// TwinCAT 3 PLC project CEFPLC
// ProgramVersion: 3.1.4022.3
// libraries:
//   Tc2_Standard, * (Beckhoff Automation GmbH)
//   Tc2_System, * (Beckhoff Automation GmbH)
//   Tc2_Utilities, * (Beckhoff Automation GmbH)
//   Tc3_Database, * (Beckhoff Automation GmbH)
//   Tc3_EventLogger, * (Beckhoff Automation GmbH)
//   Tc3_Module, * (Beckhoff Automation GmbH)
//   VisuDialogs, * (System)
//   VisuSymbols,3.5.10.0,System
// project tree:
//   DUTs/ ST_ChamberAlarm.TcDUT, ST_ProgramListStruct.TcDUT, ST_ProgramStruct.TcDUT, ST_ScheduleStruct.TcDUT
//   FB/ fbCalculateSetpoint.TcPOU, scaleValue.TcPOU
//   / GlobalTextList.TcGTLO, PlcTask.TcTTO, ST_Record.TcDUT, Visualization Manager.TcVMO (not stored), VISU_TASK.TcTTO
//   GVLs/ GVL.TcGVL, IO_VARS.TcGVL
//   POUs/ AlarmLogger.TcPOU, DeleteOldData.TcPOU, Humidity.TcPOU, HumidityPID.TcPOU, HeaterDuty.TcPOU, TempPID.TcPOU, IO.TcPOU, OkToRun.TcPOU, MAIN.TcPOU, Watering.TcPOU
//   POUs/OLD NOT USED/ POU.TcPOU, fbGetNextLine.TcPOU, fbGetNextLineAfterMidnight.TcPOU, GetPreviousLine.TcPOU
//   POUs/Program Setpoints/ DatabaseStateMachine.TcPOU, DBConnector.TcPOU, QueryProgram.TcPOU
//   POUs/Scheduing/ fbGetCurrentProgramName.TcPOU, fbGetCurrentScheduleLine.TcPOU, fbGetFirstScheduleLine.TcPOU, fbGetNextScheduleLine.TcPOU, Scheduler.TcPOU
//   VISUs/ HMI_MAIN.TcVIS, OverviewScreen.TcVIS, GraphScreen.TcVIS, Settings.TcVIS, ProgramScreen.TcVIS, ImagePool.TcIPO (not stored), ManualMode.TcVIS, IO.TcVIS, Alarms.TcVIS, Watering.TcVIS
// real-time tasks:
//   TASK PlcTask: cycle T#10ms, priority 20, ADS port 350
//   TASK VISU_TASK: cycle T#50000us, priority 30, ADS port 351
// I/O:
//   DEVICE Device 2 (EtherCAT), AmsNetId 192.168.1.102.3.1
//     Term 1 (EK1100) [EK1100 EtherCAT Coupler (2A E-Bus)]
//       Term 2 (EL1008) [EL1008 8Ch. Dig. Input 24V, 3ms]
//       Term 3 (EL2008) [EL2008 8Ch. Dig. Output 24V, 0.5A]
//       Term 4 (EL2008) [EL2008 8Ch. Dig. Output 24V, 0.5A]
//       Term 5 (EL3064) [EL3064 4Ch. Ana. Input 0-10V]
//       Term 6 (EL4002) [EL4002 2Ch. Ana. Output 0-10V, 12bit]
//       Term 7 (EL9011) [EL9011 End Terminal]
// variable links:
//   CEFPLC/CEFPLC Instance <-> Device 2 (EtherCAT)/Term 1 (EK1100)/Term 3 (EL2008)
//     PlcTask Outputs/IO_VARS.HPS1 <-> Channel 4/Output
//     PlcTask Outputs/IO_VARS.HPS2 <-> Channel 5/Output
//     PlcTask Outputs/IO_VARS.HPS3 <-> Channel 6/Output
//     PlcTask Outputs/IO_VARS.MH1 <-> Channel 1/Output
//     PlcTask Outputs/IO_VARS.MH2 <-> Channel 2/Output
//     PlcTask Outputs/IO_VARS.MH3 <-> Channel 3/Output
//   CEFPLC/CEFPLC Instance <-> Device 2 (EtherCAT)/Term 1 (EK1100)/Term 4 (EL2008)
//     PlcTask Outputs/IO_VARS.ALARM <-> Channel 5/Output
//     PlcTask Outputs/IO_VARS.AUX1 <-> Channel 1/Output
//     PlcTask Outputs/IO_VARS.AUX2 <-> Channel 2/Output
//     PlcTask Outputs/IO_VARS.AUX3 <-> Channel 3/Output
//     PlcTask Outputs/IO_VARS.ENABLE <-> Channel 7/Output
//     PlcTask Outputs/IO_VARS.HEATERS <-> Channel 4/Output
//     PlcTask Outputs/IO_VARS.HUMVALVE <-> Channel 6/Output
//   CEFPLC/CEFPLC Instance <-> Device 2 (EtherCAT)/Term 1 (EK1100)/Term 5 (EL3064)
//     PlcTask Inputs/GVL.tempSensor <-> AI Standard Channel 1/Value
//     PlcTask Inputs/GVL.tempSensor2 <-> AI Standard Channel 3/Value
//     PlcTask Inputs/IO_VARS.HUM_SENS <-> AI Standard Channel 2/Value
//     PlcTask Inputs/IO_VARS.HUM_SENS2 <-> AI Standard Channel 4/Value
//   CEFPLC/CEFPLC Instance <-> Device 2 (EtherCAT)/Term 1 (EK1100)/Term 6 (EL4002)
//     PlcTask Outputs/IO_VARS.FANSPEED <-> AO Outputs Channel 2/Analog output
//     PlcTask Outputs/IO_VARS.GLYCOL_VALVE <-> AO Outputs Channel 1/Analog output

CONFIGURATION CEFPLC
    RESOURCE PLC ON TwinCAT3
        TASK PlcTask(INTERVAL := T#10ms, PRIORITY := 20);
        TASK VISU_TASK(INTERVAL := T#50000us, PRIORITY := 30);
        PROGRAM MAIN WITH PlcTask : MAIN;
        PROGRAM VisuElems_Visu_Prg WITH VISU_TASK : VisuElems.Visu_Prg;
    END_RESOURCE
END_CONFIGURATION

// ---- DUTs/ST_ChamberAlarm.TcDUT
TYPE ST_ChamberAlarm :
STRUCT
	dtTime:STRING(255);
	sAlarmText:STRING(255);
	
	
END_STRUCT
END_TYPE

// ---- DUTs/ST_ProgramListStruct.TcDUT
TYPE ST_ProgramListStruct :
STRUCT
	ID: LINT;
	Name: STRING(255);
END_STRUCT
END_TYPE

// ---- DUTs/ST_ProgramStruct.TcDUT
{attribute 'enable_dynamic_creation'}
TYPE ST_ProgramStruct :
STRUCT
	ID: LINT;
	name: STRING(255);
	ProgramID: LINT;
	iTime: LINT;
	Temperature: LREAL;
	humidity: LREAL;
	Light1: INT;
	Light2: INT;
	DO10: BOOL;
	DO11: BOOL;
END_STRUCT
END_TYPE

// ---- DUTs/ST_ScheduleStruct.TcDUT
TYPE ST_ScheduleStruct :
STRUCT
	ID: LINT;
	Sequence: LINT;
	ProgramID: LINT;
END_STRUCT
END_TYPE

// ---- ST_Record.TcDUT
TYPE ST_Record :
STRUCT

    nID        : LINT;
    dtTimestamp: DATE_AND_TIME;
    sName      : STRING;
    nSensor1   : LREAL;
    nSensor2   : LREAL;
END_STRUCT
END_TYPE

// ---- GVLs/GVL.TcGVL
{attribute 'qualified_only'}
VAR_GLOBAL
	

	TempControl: LREAL;
	iTempControl AT %Q*:INT;
	cycleTime: LREAL;
	
	tempSensor AT %I*: INT; 
	tempSensor2 AT %I*: INT; 
	
	Temp,Temp2: LREAL;
	Humidity,Humidity2:LREAL;

	
	reset: BOOL;

	fbLocalSystemTime:FB_LocalSystemTime;

	programURL: STRING(255);
	graphURL:STRING(255);
		
	manualMode:BOOL;
	bActiveAlarm:BOOL;
	bCriticalAlarm:BOOL;
	sAlarmText:STRING(255);
	sInfoText:STRING(255);
	
	
	
END_VAR

VAR_GLOBAL PERSISTENT
	KpCooling : LREAL := 10;
	KiCooling : LREAL := 550;
	KdCooling : LREAL := 0;
	KvCooling : LREAL := 800;
	
	KpHeating : LREAL := 3000;
	KiHeating : LREAL := 550;
	KdHeating: LREAL := 0;
	KvHeating : LREAL := 320;
	
	KpHumidity : LREAL := 1;
	KiHumidity : LREAL := 1;
	KdHumidity: LREAL := 0;
	KvHumidity : LREAL := 1;
	
	CurrentProgram: LINT;
	CurrentProgramName:STRING(255);
	NextProgram: LINT;
	FirstProgram:LINT;
	ScheduleSequence:LINT;

	TempAlarmHigh:LREAL:=50;
	TempAlarmLow:LREAL:=4;
	
	TempCalibrationLimit:REAL:=10;//in percent
	HumCalibrationLimit:REAL:=10;//in percent
	//Don't change this without also changing
	//iMax in AlarmLogger
	aAlarms:ARRAY[0..15] OF ST_ChamberAlarm;
	
	okToRun:BOOL;
	iState:INT;
	
	
	
	//Setpoint variable declariations
	Light1Max:INT:=2; //Max light level
	Light1Level:INT; //Current light level
	Light1Percent:REAL; //Current light level in percent of max
	Light1Stepmode:BOOL;
	
	Light2Max:INT:=2; //Max light level
	Light2Level:INT; //Current light level
	Light2Percent:REAL; //Current light level in percent of max
	Light2Stepmode:BOOL;
	
	TempSetpoint: LREAL;
	TempStepmode: BOOL;
	
	HumiditySetpoint:LREAL;
	HumidityStepmode:BOOL;
	
	
	///HMI VARS
	HMIPowerButton:BOOL;
	HMIFanSpeed:INT;
	HMIWateringStartHour:DWORD;
	HMIWateringStartMinute:DWORD;
	HMIWateringTimeSeconds:DWORD;
	
	//Watering
	wateringDays: ARRAY[0..6] OF BOOL; //if element 0 is True, then water on Sunday, if element 1 is true, water on Monday. etc
	watertingTime:TIME;//How long to water
	watertingStart:TOD;//When to start watering
END_VAR

// ---- GVLs/IO_VARS.TcGVL
{attribute 'qualified_only'}
VAR_GLOBAL
	
PRESSURE_SENSE AT %I*:BOOL;
HUM_SENS,HUM_SENS2 AT %I*:INT;


ENABLE AT %Q*:BOOL;
MH1,MH2,MH3 AT %Q*:BOOL;
HPS1,HPS2,HPS3 AT %Q*:BOOL;
AUX1,AUX2,AUX3,ALARM AT %Q*:BOOL; 
HEATERS AT %Q*:BOOL;

HUMVALVE AT %Q*:BOOL;

GLYCOL_VALVE AT %Q*:INT;

END_VAR

VAR_GLOBAL PERSISTENT
	FANSPEED AT %Q*:INT;
END_VAR

// ---- POUs/MAIN.TcPOU
PROGRAM MAIN


VAR

	GETCPUCOUNTER: GETCPUCOUNTER; //CPU tick function block definition
	previous_low_ticks,low_ticks,high_ticks: UDINT; //Vars to hold the cpu tick count
	
	
	test: DINT; //I don't know what this is
	sqlResult : WSTRING(255);//I don't think we need this anymore either
	bsqlError: BOOL;//same ehere
	
	numberOfLinesOut: LINT; //and here
	Scaled_control: LREAL;//this moved too

	fbTON: TON := (PT := TIME#1S0MS); //PID TON TIMER.
	restartTime: TON := (PT := TIME#60S0MS);//AUTO RESTART TIMER

	

	getHost: FB_GetHostName; //Get host name function block definition
	myName: STRING(255); //Var to hold host name. If the host name is more than 255 chars you're doing something wrong.
	
	FB_WritePersistentData: FB_WritePersistentData;
	GETSYSTEMTIME:GETSYSTEMTIME;
END_VAR

/////////////////////////////////////////////////////////////
//CALCULATE CYCLE TIME FOR PLC
previous_low_ticks := low_ticks;
//GETCPUCOUNTER(cpuCntLoDW=> low_ticks, cpuCntHiDW=> high_ticks);
GETSYSTEMTIME(timeLoDW=> low_ticks, timeHiDW=> high_ticks);
//low ticks is a 64 bit int and rolls over into high ticks once in a while. So we make sure we're not calculating the overflow
IF previous_low_ticks < low_ticks THEN 
	GVL.cycleTime := UDINT_TO_LREAL(low_ticks-previous_low_ticks)*0.000000100;//Each tick is 100ns
END_IF

/////////////////////////////////////////////////////////////
//GET HOST NAME AND CONCAT URLS FOR HMI SCREENS
//we need the hostname because "localhost" doesn't work if
//you're connected remotely, duh
getHost(bExecute:= TRUE, sHostName=>myName );
GVL.programURL:=CONCAT('http://',myName);
GVL.programURL:=CONCAT(GVL.programURL,':8050');
GVL.graphURL:=CONCAT('http://',myName);
GVL.graphURL:=CONCAT(GVL.graphURL,':8050/graph');
/////////////////////////////////////////////////////////////
//VARIOUS PROGRAMS THAT NEED TO RUN EVERY CYCLE
IO(); //Input/Output tasks and calculations
Humidity();
HeaterDuty();
OkToRun();//Alarms
fbTON();//Timer for some functions that we don't want to run every cycle
restartTime();//Timer for auto restart in the event of an error. Set to 60 seconds
AlarmLogger();//Log alarms (if any)
GVL.fbLocalSystemTime(sNetID:= '', bEnable:= TRUE, dwCycle:= 1);//Get the current date and time

/////////////////////////////////////////////////////////////
//VARIOUS PROGRAMS THAT DO NOT RUN EVERY CYCLE

IF fbTON.Q=TRUE THEN //when the timer is true (every 1 second)
	TempPID();//Run the PIDs
	HumidityPID();
	fbTON.IN:=FALSE; //reset the timer
	FB_WritePersistentData(NETID:='', PORT:=851, START:=TRUE, TMOUT:=T#1S ); //Write persistent data 
	Scheduler();//Checking/setting program schedule
	DeleteOldData();
	Watering();
ELSE
	fbTON.IN:=TRUE; //If the timer is not true...keep timing until it is!
END_IF
/////////////////////////////////////////////////////////////
//MAIN STATE MACHINE
CASE GVL.iState OF
	//STARTUP
	0:
		
		GVL.reset:=TRUE; //RESET THE PID MEMORY BEFORE STARTING. THIS IS IMPORTANT.
		Scheduler.resetSchedule:=TRUE; //RESET THE SCHEDULE BACK TO THE BEGINNING 
		
		IF GVL.sInfoText='' THEN//If the info text is blank, give the user a hint to get started
			GVL.sInfoText:='Setup programs & settings then Start';
		END_IF
		//Check if user presses start button	
		IF GVL.HMIPowerButton=TRUE THEN

			DatabaseStateMachine.bStepStart:=TRUE; //STEP START MEANS THE FIRST SETPOINT WILL BE STEPPED TO GET STARTED. MORE INFO IN DOCS
			DatabaseStateMachine(); //ALL SETPOINTS ARE CONTROLLED BY THE DATABASE STATE MACHINE. THIS PROGRAM IS IMPORTANT.
			
			GVL.sAlarmText:='Wait for Startup...';
			GVL.sInfoText:='Checking Setpoints...';
			IF DatabaseStateMachine.allOutputsSet=TRUE AND GVL.okToRun=TRUE THEN //Once everything is set, we can move on to the next state
				GVL.iState:=1;
				
			END_IF
	
		END_IF
		
		IF GVL.manualMode THEN
			GVL.iState:=254;
		END_IF
	
	1:
		//Runninng

		GVL.reset:=FALSE; //Don't reset the PID while running
		
		DatabaseStateMachine.bStepStart:=FALSE;//Don't need step start because we're already running!
		DatabaseStateMachine();//Running the statemachine....
		GVL.sInfoText:=''; //Everything is good! We don't need any info text
		
		//Check if shutdown
		//Lots of things can make OktoRun False. Check the sub program and the Docs.
		IF GVL.okToRun=FALSE THEN 
			GVL.iState:=2;
		END_IF
		
	2:
	//Shutdown
	
	IF GVL.bCriticalAlarm=FALSE THEN //If shutdown with no error
		
		GVL.iState:=0;

		
	ELSIF GVL.bCriticalAlarm=TRUE THEN//If shutdown WITH error

		restartTime.IN:=TRUE;
		GVL.sInfoText:='Acknowledge alarm or wait for auto restart';
		IF restartTime.Q THEN //Try restarting after the timer has elapsed
			GVL.HMIPowerButton:=TRUE;
			GVL.bCriticalAlarm:=FALSE;
			restartTime.IN:=FALSE;
			GVL.iState:=1;
			GVL.sInfoText:='Error occured...restarting';
		ELSIF GVL.bActiveAlarm=FALSE THEN //Clear error if the user has pressed the acknowledge alarm button
			restartTime.IN:=FALSE;
			GVL.bCriticalAlarm:=FALSE;
			GVL.iState:=0;
			GVL.sInfoText:='Alarm acknowledged, please manually restart program ';
		END_IF

	END_IF
	254:
	//Manual Mode
	//Just don't do anything until the user exits manual mode
		GVL.sAlarmText:='MANUAL MODE ACTIVE';
		IF GVL.manualMode=FALSE THEN
			GVL.iState:=2;
		END_IF
	
END_CASE

END_PROGRAM

// ---- POUs/IO.TcPOU
PROGRAM IO
VAR


	Scaled_control: LREAL;

END_VAR


	

GVL.Temp := 0.010071*INT_TO_LREAL(GVL.tempSensor) - 39.996;//See documentation for sensor
GVL.Humidity := (INT_TO_LREAL(IO_VARS.HUM_SENS)/3.2767)*100/5000;

GVL.Temp2 := 0.010071*INT_TO_LREAL(GVL.tempSensor2) - 39.996;//See documentation for sensor
GVL.Humidity2 := (INT_TO_LREAL(IO_VARS.HUM_SENS2)/3.2767)*100/5000;

IO_VARS.ALARM:=GVL.bCriticalAlarm;//alarm buzzer


//Check this variable just to make sure we don't break anything
IF GVL.HMIFanSpeed>100 THEN
	GVL.HMIFanSpeed:=100;
END_IF

IF GVL.HMIFanSpeed<0 THEN
	GVL.HMIFanSpeed:=0;
END_IF

IO_VARS.FANSPEED := REAL_TO_INT(16384*-50*LOG(0.00001*(63949-630*GVL.HMIFanSpeed))/100);//Scaling. outout is nonlinear for this board. Equation is x = -50 log(.00001(63949 - 630 y))
	
IF IO_VARS.FANSPEED>16385 THEN
	IO_VARS.FANSPEED:=16385;//DO NOT EXCEED 5 VOLTS FOR THAT CONTROL BOARD
END_IF

IF IO_VARS.FANSPEED<3276 THEN
	IO_VARS.FANSPEED:=3276;//IT'S DANGERIOUS TO RUN THE CHAMBER WITH THE FANS COMPLETELY OFF
END_IF


IF GVL.manualMode=FALSE THEN
	
	//Set the valve state
	IO_VARS.GLYCOL_VALVE:=GVL.iTempControl;
	
	IO_VARS.AUX1:=Watering.waterOn;//Watering bound to aux 1
	
	//If the output of the pulse timer is true, turn on the heater valve
	IO_VARS.HEATERS:=HeaterDuty.HeatersON;
	
	//If the output of the pulse timer is true, turn on the humidity valve
	IO_VARS.HUMVALVE:=Humidity.HumidityON;
		
	////////////MAPPING METAL HALIDE LIGHTS/////////////
	IF GVL.Light1Level=0 THEN
		IO_VARS.MH1:=0;
		IO_VARS.MH2:=0;
		IO_VARS.MH3:=0;
	ELSIF  GVL.Light1Level=1 THEN
		IO_VARS.MH1:=1;
		IO_VARS.MH2:=0;
		IO_VARS.MH3:=0;
	ELSIF  GVL.Light1Level=2 THEN
		IO_VARS.MH1:=1;
		IO_VARS.MH2:=1;
		IO_VARS.MH3:=0;
	ELSIF  GVL.Light1Level=3 THEN
		IO_VARS.MH1:=1;
		IO_VARS.MH2:=1;
		IO_VARS.MH3:=1;
	END_IF
	
	////////////MAPPING HIGH PRESSURE SODIUM LIGHTS/////////////
	IF GVL.Light2Level=0 THEN
		IO_VARS.HPS1:=0;
		IO_VARS.HPS2:=0;
		IO_VARS.HPS3:=0;
	ELSIF  GVL.Light2Level=1 THEN
		IO_VARS.HPS1:=1;
		IO_VARS.HPS2:=0;
		IO_VARS.HPS3:=0;
	ELSIF  GVL.Light2Level=2 THEN
		IO_VARS.HPS1:=1;
		IO_VARS.HPS2:=1;
		IO_VARS.HPS3:=0;
	ELSIF  GVL.Light2Level=3 THEN
		IO_VARS.HPS1:=1;
		IO_VARS.HPS2:=1;
		IO_VARS.HPS3:=1;
	END_IF
	
END_IF

END_PROGRAM

// ---- POUs/Humidity.TcPOU
PROGRAM Humidity
VAR
	
	fbTON: TON; // TON TIMER.
	
	fbTP: TP;

	pulseDuration: TIME:=TIME#2S;
END_VAR

VAR_OUTPUT
	
HumidityON:BOOL;
	


END_VAR

//This program pulses the humidity for a certain number of seconds based on the PID output

//This timer determines how often to pulse, and the max length of the pulse
//In other words, we're making a Duty Cycle
fbTON(PT := TIME#30S0MS);

//Run the pulse timer
fbTP();

//If the output of the pulse timer is true, turn on the humidity valve
HumidityON:=fbTP.Q;


//Don't worry about negative values
IF HumidityPID.output >=0 THEN
	
	//Convert the output to a time (in milliseconds)
	pulseDuration:=LREAL_TO_TIME(HumidityPID.output);
	
	//Don't pulse anything shorter than 500ms.
	//It's bad for the relay & valve
	IF pulseDuration<TIME#500MS THEN
		pulseDuration:=TIME#0MS;
	END_IF
	
	//If the durataion is greater than the max duration
	//Just turn it on and leave it on
	IF pulseDuration>fbTON.PT THEN
		HumidityON:=TRUE;
	ELSE
	
		IF fbTON.Q=TRUE THEN //when the timer is true 
			fbTP(IN:=TRUE, PT:=pulseDuration);//set the pulse length
			fbTON.IN:=FALSE;//Reset the timer funtion
		ELSE
			fbTON.IN:=TRUE; //If the timer is not true...keep timing until it is!
			fbTP.IN:=FALSE;//reset the pulse function
		END_IF
			
	END_IF

END_IF

END_PROGRAM

// ---- POUs/HumidityPID.TcPOU
PROGRAM HumidityPID
VAR
	
	PID: FB_BasicPID;
	bReset: BOOL;
	
	AH: LREAL;
	AHSetpoint: LREAL;
	
	//Constants for air as an ideal gas to calculate absolute humidity in g/m^3
	Tn:LREAL:=240.7263;
	m:LREAL:=7.591386;
	A:LREAL:=6.116441;
END_VAR

VAR_OUTPUT
	output: LREAL;
END_VAR

//Convert realative humidity to absolute humidity in grams per cubic meter
AH:= A*EXPT	(10,m*GVL.Temp/(GVL.Temp+Tn))*(GVL.Humidity/100)*100*2.16679/(273.15+GVL.Temp);
AHSetpoint:= A*EXPT(10,m*GVL.TempSetpoint/(GVL.TempSetpoint+Tn))*(GVL.HumiditySetpoint/100)*100*2.16679/(273.15+GVL.TempSetpoint);

//Run pid loop
PID(
	fSetpointValue:=AHSetpoint,
	fActualValue:=AH, 
	bReset:=bReset, 
	fCtrlCycleTime:=1, 
	fKp:=GVL.KpHumidity, 
	fTn:=GVL.KiHumidity, 
	fTv:=GVL.KvHumidity, 
	fTd:=GVL.KdHumidity, 
	fCtrlOutput=>output);
	
	
//Since there's no dehumidification on this chamber
//Just reset the PID back to 0 if the output is negative
IF output<0 THEN
	output:=0;
	bReset:=TRUE;
ELSIF GVL.reset =  TRUE THEN
	bReset:=TRUE;
ELSE
	bReset:=FALSE;
END_IF

END_PROGRAM

// ---- POUs/Watering.TcPOU
PROGRAM Watering
VAR
	
	trigger:F_TRIG;
	waterTimer:TON;
	waterOn:BOOL;
	dtTime:DT;
	todTime:TOD;

END_VAR


GVL.watertingTime:=DWORD_TO_TIME(GVL.HMIWateringTimeSeconds*1000);//in ms
GVL.watertingStart:=DWORD_TO_TOD((GVL.HMIWateringStartHour*60 + GVL.HMIWateringStartMinute)*60*1000);//also in ms



dtTime:=SYSTEMTIME_TO_DT(GVL.fbLocalSystemTime.systemTime);
todTime:=DT_TO_TOD(dtTime);
waterTimer(PT:=GVL.watertingTime);

IF GVL.wateringDays[GVL.fbLocalSystemTime.systemTime.wDayOfWeek]=TRUE THEN
	IF todTime>=GVL.watertingStart AND todTime<=(GVL.watertingStart+GVL.watertingTime) THEN
		waterOn:=TRUE;
	ELSE
		waterOn:=FALSE;
	END_IF
END_IF

END_PROGRAM

// ---- POUs/HeaterDuty.TcPOU
PROGRAM HeaterDuty
VAR
	
	fbTON: TON; // TON TIMER.
	
	fbTP: TP;

	pulseDuration: TIME:=TIME#2S;
END_VAR

VAR_OUTPUT
	
HeatersON:BOOL;
	
END_VAR

//This program pulses the heaters for a certain number of seconds based on the PID output

//This timer determines how often to pulse, and the max length of the pulse
//In other words, we're making a Duty Cycle
fbTON(PT := TIME#30S0MS);

//Run the pulse timer
fbTP();

//If the output of the pulse timer is true, turn on the heater valve
HeatersON:=fbTP.Q;


//Don't worry about negative values
IF TempPID.HeatingOutput >=0 THEN
	
	//Convert the output to a time (in milliseconds)
	pulseDuration:=LREAL_TO_TIME(TempPID.HeatingOutput);
	
	//Don't pulse anything shorter than 500ms.
	//It's bad for the relay
	IF pulseDuration<TIME#500MS THEN
		pulseDuration:=TIME#0MS;
	END_IF
	
	//If the durataion is greater than the max duration
	//Just turn it on and leave it on
	IF pulseDuration>fbTON.PT THEN
		HeatersON:=TRUE;
	ELSE
	
		IF fbTON.Q=TRUE THEN //when the timer is true 
			fbTP(IN:=TRUE, PT:=pulseDuration);//set the pulse length
			fbTON.IN:=FALSE;//Reset the timer funtion
		ELSE
			fbTON.IN:=TRUE; //If the timer is not true...keep timing until it is!
			fbTP.IN:=FALSE;//reset the pulse function
		END_IF
			
	END_IF

END_IF

END_PROGRAM

// ---- POUs/TempPID.TcPOU
PROGRAM TempPID
VAR
	
	PIDCooling: FB_BasicPID;
	PIDHeating: FB_BasicPID;
	bResetCooling: BOOL;
	bResetHeat: BOOL;
END_VAR

VAR_OUTPUT
	CoolingOutput: LREAL;
	HeatingOutput: LREAL;
END_VAR



//Run pid loop
PIDCooling(
	fSetpointValue:=GVL.TempSetpoint,
	fActualValue:=GVL.Temp, 
	bReset:=bResetCooling, 
	fCtrlCycleTime:=1, 
	fKp:=GVL.KpCooling, 
	fTn:=GVL.KiCooling, 
	fTv:=GVL.KvCooling, 
	fTd:=GVL.KdCooling);



PIDHeating(
	fSetpointValue:=GVL.TempSetpoint,
	fActualValue:=GVL.Temp, 
	bReset:=bResetHeat, 
	fCtrlCycleTime:=1, 
	fKp:=GVL.KpHeating, 
	fTn:=GVL.KiHeating, 
	fTv:=GVL.KvHeating, 
	fTd:=GVL.KdHeating);
	
//Reset the PID back to 0 if the output is out of range
IF  PIDCooling.fCtrlOutput>50 THEN
	bResetCooling:=TRUE;
ELSIF GVL.reset =  TRUE THEN
	bResetCooling:=TRUE;
ELSE
	bResetCooling:=FALSE;
	CoolingOutput:=PIDCooling.fCtrlOutput*-105+14089; //<----important scaling function because the old staefa valves are weird. See documentation for siemens ZM-101A
END_IF

//Reset the PID back to 0 if the output is out of range
IF PIDHeating.fCtrlOutput<-30000 THEN
	bResetHeat:=TRUE;
ELSIF GVL.reset =  TRUE THEN
	bResetHeat:=TRUE;
ELSE
	bResetHeat:=FALSE;
	HeatingOutput:=PIDHeating.fCtrlOutput;//No need to scale the heater output. Just use PID constants
END_IF

//If there is more than 5% cooling demand, turn off the heaters completely. (i.e. don't waste energy)
IF PIDCooling.fCtrlOutput<-5 THEN
	HeatingOutput:=0;
END_IF

//Scale temp signal for analog out to avoid overflows/negative numbers
IF CoolingOutput>=32767 THEN
	GVL.iTempControl :=32767;
ELSIF CoolingOutput <=0 THEN
	GVL.iTempControl :=0;
ELSE
	GVL.iTempControl := LREAL_TO_INT(CoolingOutput);
END_IF

IF HeatingOutput>=30000 THEN
	HeatingOutput :=30000;
ELSIF HeatingOutput <=0 THEN
	HeatingOutput :=0;
ELSE
	HeatingOutput := HeatingOutput;
END_IF

END_PROGRAM

// ---- POUs/OkToRun.TcPOU
PROGRAM OkToRun
VAR

	alarmTimeout: TON := (PT := TIME#11S0MS);
	
END_VAR

alarmTimeout();

//HARD CODED UPPER AND LOWER LIMITS
IF GVL.Temp > 50 THEN
		GVL.bCriticalAlarm:=TRUE;
		IO_VARS.ENABLE:=FALSE;
		GVL.sAlarmText:='Critical High Temp Alarm';
	END_IF
IF GVL.Temp < 0 THEN
	GVL.bCriticalAlarm:=TRUE;
	IO_VARS.ENABLE:=FALSE;
	GVL.sAlarmText:='Critical Low Temp Alarm';
END_IF



//If not in manual mode
IF GVL.manualMode=FALSE THEN
	
	//If running
	IF GVL.iState=1 THEN

	
		//Temperature Alarm Logic for STEP MODE
		IF GVL.TempStepmode THEN
			IF GVL.iState=1 AND GVL.Temp > (GVL.TempAlarmHigh) THEN
				GVL.bCriticalAlarm:=TRUE;
				GVL.sAlarmText:='High Temp Alarm';
			END_IF
			IF GVL.iState=1 AND GVL.Temp < (GVL.TempAlarmLow) THEN
				GVL.bCriticalAlarm:=TRUE;
				GVL.sAlarmText:='Low Temp Alarm';
			END_IF
		END_IF
		
		//Temperature alarm logic for RAMP MODE
		IF GVL.TempStepmode=FALSE THEN
			IF GVL.iState=1 AND GVL.Temp > (GVL.TempSetpoint+GVL.TempAlarmHigh) THEN
				GVL.bCriticalAlarm:=TRUE;
				GVL.sAlarmText:='High Temp Alarm';
			END_IF
			IF GVL.iState=1 AND GVL.Temp < (GVL.TempSetpoint-GVL.TempAlarmLow) THEN
				GVL.bCriticalAlarm:=TRUE;
				GVL.sAlarmText:='Low Temp Alarm';
			END_IF
		END_IF
		
		//Schedule Alarms
		//If the user deletes the current program or changes the schedule in an incorrect way, 
		//Tell them they messed up
		//This could also happen if there are database errors
		IF fbGetCurrentScheduleLine.sSeverity="No Error" AND fbGetCurrentScheduleLine.iLines=0 THEN
			alarmTimeout.IN:=TRUE;
			IF alarmTimeout.Q=TRUE THEN
				GVL.sAlarmText:='Error getting current program. Check schedule and programs';
				GVL.bCriticalAlarm:=TRUE;
				alarmTimeout.IN:=FALSE;
				
			END_IF
				
		ELSE

			alarmTimeout.IN:=FALSE;
			
		END_IF
		//Temperature sensor alarm
		IF ABS((GVL.Temp-GVL.Temp2)*100/GVL.Temp)>GVL.TempCalibrationLimit THEN
				GVL.sAlarmText:='Temperature Sensor Error.';
				GVL.bCriticalAlarm:=TRUE;
		END_IF
		
		//Humidity sensor alarm
		IF ABS((GVL.Humidity-GVL.Humidity2)*100/GVL.Humidity)>GVL.HumCalibrationLimit THEN
				GVL.sAlarmText:='Humidity Sensor Error.';
				GVL.bCriticalAlarm:=TRUE;
		END_IF
		

	END_IF
	
	

END_IF	

//OK TO RUN IF THERE ARE NO ERRORS
IF GVL.bCriticalAlarm=FALSE AND GVL.HMIPowerButton=TRUE THEN
	GVL.okToRun:=TRUE;
	GVL.sAlarmText:='Running No Alarm';
	IO_VARS.ENABLE:=TRUE;
ELSIF GVL.bCriticalAlarm=FALSE AND GVL.HMIPowerButton=FALSE AND IO_VARS.ENABLE=FALSE THEN
	GVL.sAlarmText:='Not Running No Alarm';
ELSE
	GVL.okToRun:=FALSE;
	IF GVL.manualMode=FALSE THEN
		IO_VARS.ENABLE:=FALSE;
	END_IF
	
	GVL.HMIPowerButton:=FALSE;
END_IF

END_PROGRAM

// ---- POUs/Scheduing/fbGetCurrentScheduleLine.TcPOU
PROGRAM fbGetCurrentScheduleLine

VAR_OUTPUT
	arrRecords: ST_ScheduleStruct;
	sSeverity: WSTRING(255);
	bError :BOOL;

	iLines: UDINT;
END_VAR
VAR
	STProgram: ST_ProgramStruct;
	now : TIMESTRUCT;
	nowMinutes : LINT;
	
	previousMinute: LINT;
	
	fbTON: TON := (PT := TIME#10S0MS);

	

	
	fbPLCDBRead : FB_PLCDBRead(sNetID:='',tTimeout:=T#5S);
	fbSqlCommand : FB_SQLCommand(sNetID := '', tTimeout := T#5S);
	
	
	intTime: DINT;
	todTime: TOD;

	sCmd: STRING(255):='SELECT * FROM [Schedule] ORDER BY [Sequence] ASC';

	dIntSqlResult: DINT;
	fbSQLDatabase: FB_SQLDatabase(sNetID:='', tTimeout:=T#10S);
	fbSQLResult: FB_SQLResult(sNetID:='', tTimeout:=T#10S);
	result: I_TcResultEvent;


	iState: INT;
END_VAR

//Build command



sCmd :=CONCAT('SELECT * FROM [Schedule] WHERE [Sequence]=',LINT_TO_STRING(GVL.ScheduleSequence));

//State machine
CASE iState OF
0:
//IDLE
fbTON(PT := TIME#3S0MS);
IF fbTON.Q=TRUE THEN
	iState:=1;
	fbTON.IN:=FALSE;
	bError := FALSE; 
ELSE
	fbTON.IN:=TRUE;
END_IF
//Connect
1:
	IF fbSqlDatabase.Connect(1) THEN
		IF fbSqlDatabase.bError THEN
			iState := 255;
			result := fbSqlDatabase.ipTcResultEvent;
			sSeverity := result.Text;
			bError := TRUE; 		
		ELSE
			//If sucessful, point the connection to the sql command function
			fbSqlDatabase.CreateCmd(ADR(fbSqlCommand));
			iState := 2;
		END_IF
	END_IF
2:
//Send the sql command
	IF fbSQLCommand.ExecuteDataReturn(ADR(sCmd), SIZEOF(sCmd), ADR(fbSqlResult)) THEN
		IF fbSQLCommand.bError THEN
			iState := 255;
			result := fbSQLCommand.ipTcResultEvent;
			sSeverity := result.Text;
			bError := TRUE;
		ELSE
			iState := 3; 
			iLines:=fbSqlResult.nDataCount;
		END_IF
	END_IF
		
3:
//Read the sql result
	IF fbSqlResult.Read(0, 1, ADR(arrRecords), SIZEOF(arrRecords), TRUE, TRUE) THEN
		IF fbSqlResult.bError THEN
			result := fbSqlResult.ipTcResultEvent;
			sSeverity := result.Text;
			iState:=255;
			bError := TRUE;
		ELSE 
			iState:=4;
			
			result := fbSqlResult.ipTcResultEvent;
			sSeverity := result.Text;
		END_IF
	

	END_IF
4:
	IF 	fbSqlDatabase.Disconnect() THEN
		bError := FALSE;
		iState:=0;
	END_IF
255:
	IF 	fbSqlDatabase.Disconnect() THEN
		iState:=0;	
		bError := TRUE;
		result := fbSqlResult.ipTcResultEvent;
		sSeverity := result.Text;

	END_IF
	
END_CASE

END_PROGRAM

// ---- POUs/AlarmLogger.TcPOU
PROGRAM AlarmLogger
VAR
	iCounter:DINT;
	iMax:DINT;
	alarmTrigger: R_TRIG; 
END_VAR

alarmTrigger(CLK := GVL.bCriticalAlarm);

IF alarmTrigger.Q THEN
	//Shift the whole array by 1 so we can enter the new alarm in the first element
	iCounter:=0;
	
	//Max number of alarms
	//Depends on the array size of GVL.aAlarms
	iMax:=15;
	
	FOR iCounter:=iMax TO 0 BY -1 DO //Notice we're counting backwards so the last element goes away, and the first element is now empty
		
		IF iCounter<>iMax THEN
			GVL.aAlarms[iCounter+1]:=GVL.aAlarms[iCounter];
		END_IF	

	END_FOR

	GVL.aAlarms[0].sAlarmText:=GVL.sAlarmText;
	GVL.aAlarms[0].dtTime:=SYSTEMTIME_TO_STRING(GVL.fbLocalSystemTime.systemTime);
	
	GVL.bActiveAlarm:=TRUE; //An alarm is now active and will remain that way until the user acknowledges it

END_IF

END_PROGRAM

// ---- POUs/Scheduing/Scheduler.TcPOU
PROGRAM Scheduler
VAR_INPUT
	resetSchedule:BOOL:=TRUE;
END_VAR
VAR
	
	
	
	ScheduleLine:ST_ScheduleStruct;
	sqlResult:WSTRING(255);
	bError:BOOL;
	iLines:UDINT;
	iState:INT;

	lastDate: TIMESTRUCT;
END_VAR


//Run all these programs to get the next line, first line, and current line in the schedule using database queries
fbGetNextScheduleLine();
fbGetCurrentScheduleLine();
fbGetFirstScheduleLine();
fbGetCurrentProgramName();
GVL.CurrentProgramName:=fbGetCurrentProgramName.arrRecords.Name;

CASE iState OF

0:
iState:=1;
//IDLE...nothing here yet

	
1:
	//If we want to reset the schedule to the beginning
	IF resetSchedule=TRUE THEN
		
		
		IF fbGetFirstScheduleLine.sSeverity="No Error" THEN //If there is no error when we try and get the first line in the schedule
			GVL.CurrentProgram:=fbGetFirstScheduleLine.arrRecords.ProgramID;
			//We need to initialize the next program to something. So we just set it to the current program
			GVL.NextProgram:=fbGetFirstScheduleLine.arrRecords.ProgramID;
			//The sequence is an integer that determines the order to run the programs. 1->2-->3 etc
			//This is set by the user in the interface. Here we just read the value
			GVL.ScheduleSequence:=fbGetFirstScheduleLine.arrRecords.Sequence;
			
			//OK we reset the schedule, set that to false now
			resetSchedule:=FALSE;
			
			//Timestamp when it happened so we know when a full day has passed
			lastDate := GVL.fbLocalSystemTime.systemTime;
		END_IF
	ELSIF resetSchedule=FALSE THEN
		//Check for the current and next programs in the schedule
		
		//While running, check to see if the schedule has changed
		//If the schedule has changed, then change the program to match
		IF fbGetCurrentScheduleLine.arrRecords.ProgramID<>GVL.CurrentProgram AND fbGetCurrentScheduleLine.sSeverity="No Error" AND fbGetCurrentScheduleLine.iLines<>0	THEN
			GVL.CurrentProgram:=fbGetCurrentScheduleLine.arrRecords.ProgramID;
		
		END_IF
		//Also get the next program
		IF fbGetNextScheduleLine.sSeverity="No Error" AND fbGetNextScheduleLine.iLines>0 THEN
			GVL.NextProgram:=fbGetNextScheduleLine.arrRecords.ProgramID;
		//If there are no more programs in the schedule, the next program will be the first program.
		ELSIF fbGetNextScheduleLine.sSeverity="No Error" AND fbGetNextScheduleLine.iLines=0 THEN
			GVL.NextProgram:=fbGetFirstScheduleLine.arrRecords.ProgramID;
		END_IF
		
		//Check if a date change has occured. 
		//We assume time always goes forward. But if the user changes the system date for some reason, this could get weird.
		IF GVL.fbLocalSystemTime.systemTime.wDay<>lastDate.wDay THEN
			//Does the next program exist? or have we reached the end of the schedule?
			IF fbGetnextScheduleLine.iLines >0 AND fbGetnextScheduleLine.sSeverity="No Error" THEN
				GVL.CurrentProgram := fbGetnextScheduleLine.arrRecords.ProgramID;
				GVL.ScheduleSequence := fbGetnextScheduleLine.arrRecords.Sequence;
				lastDate := GVL.fbLocalSystemTime.systemTime;
			ELSIF fbGetnextScheduleLine.iLines=0 AND fbGetnextScheduleLine.sSeverity="No Error" THEN
				resetSchedule:=TRUE;
				lastDate := GVL.fbLocalSystemTime.systemTime;
			END_IF
			
		END_IF
		
		
		
		
	END_IF


END_CASE

END_PROGRAM

// ---- POUs/Scheduing/fbGetNextScheduleLine.TcPOU
PROGRAM fbGetNextScheduleLine

VAR_OUTPUT
	arrRecords: ST_ScheduleStruct;
	sSeverity: WSTRING(255);
	bError :BOOL;

	iLines: UDINT;
END_VAR
VAR
	STProgram: ST_ProgramStruct;
	now : TIMESTRUCT;
	nowMinutes : LINT;
	
	previousMinute: LINT;
	
	fbTON: TON := (PT := TIME#10S0MS);

	

	
	fbPLCDBRead : FB_PLCDBRead(sNetID:='',tTimeout:=T#5S);
	fbSqlCommand : FB_SQLCommand(sNetID := '', tTimeout := T#5S);
	
	
	intTime: DINT;
	todTime: TOD;

	sCmd: STRING(255):='SELECT * FROM [Schedule] ORDER BY [Sequence] ASC';

	dIntSqlResult: DINT;
	fbSQLDatabase: FB_SQLDatabase(sNetID:='', tTimeout:=T#10S);
	fbSQLResult: FB_SQLResult(sNetID:='', tTimeout:=T#10S);
	result: I_TcResultEvent;


	iState: INT;
END_VAR

//Build command



sCmd :=CONCAT('SELECT * FROM [Schedule] WHERE [Sequence]>',LINT_TO_STRING(GVL.ScheduleSequence));

sCmd:= CONCAT(sCMD,' ORDER BY [Sequence] ASC');

//State machine
CASE iState OF
0:
//IDLE
fbTON(PT := TIME#5S0MS);
IF fbTON.Q=TRUE THEN
	iState:=1;
	fbTON.IN:=FALSE;
	bError := FALSE; 
ELSE
	fbTON.IN:=TRUE;
END_IF
//Connect
1:
	IF fbSqlDatabase.Connect(1) THEN
		IF fbSqlDatabase.bError THEN
			iState := 255;
			result := fbSqlDatabase.ipTcResultEvent;
			sSeverity := result.Text;
			bError := TRUE; 		
		ELSE
			//If sucessful, point the connection to the sql command function
			fbSqlDatabase.CreateCmd(ADR(fbSqlCommand));
			iState := 2;
		END_IF
	END_IF
2:
//Send the sql command
	IF fbSQLCommand.ExecuteDataReturn(ADR(sCmd), SIZEOF(sCmd), ADR(fbSqlResult)) THEN
		IF fbSQLCommand.bError THEN
			iState := 255;
			result := fbSQLCommand.ipTcResultEvent;
			sSeverity := result.Text;
			bError := TRUE;
		ELSE
			iState := 3; 
			iLines:=fbSqlResult.nDataCount;
		END_IF
	END_IF
		
3:
//Read the sql result
	IF fbSqlResult.Read(0, 1, ADR(arrRecords), SIZEOF(arrRecords), TRUE, TRUE) THEN
		IF fbSqlResult.bError THEN
			result := fbSqlResult.ipTcResultEvent;
			sSeverity := result.Text;
			iState:=255;
			bError := TRUE;
		ELSE 
			iState:=4;
			
			result := fbSqlResult.ipTcResultEvent;
			sSeverity := result.Text;
		END_IF
	

	END_IF
4:
	IF 	fbSqlDatabase.Disconnect() THEN
		bError := FALSE;
		iState:=0;
	END_IF
255:
	IF 	fbSqlDatabase.Disconnect() THEN
		iState:=0;	
		bError := TRUE;
		result := fbSqlResult.ipTcResultEvent;
		sSeverity := result.Text;

	END_IF
	
END_CASE

END_PROGRAM

// ---- POUs/Scheduing/fbGetFirstScheduleLine.TcPOU
PROGRAM fbGetFirstScheduleLine

VAR_OUTPUT
	arrRecords: ST_ScheduleStruct;
	sSeverity: WSTRING(255);
	bError :BOOL;

	iLines: UDINT;
END_VAR
VAR
	STProgram: ST_ProgramStruct;
	now : TIMESTRUCT;
	nowMinutes : LINT;
	
	previousMinute: LINT;
	
	fbTON: TON := (PT := TIME#10S0MS);

	

	
	fbPLCDBRead : FB_PLCDBRead(sNetID:='',tTimeout:=T#5S);
	fbSqlCommand : FB_SQLCommand(sNetID := '', tTimeout := T#5S);
	
	
	intTime: DINT;
	todTime: TOD;

	sCmd: STRING(255):='SELECT * FROM [Schedule] ORDER BY [Sequence] ASC';

	dIntSqlResult: DINT;
	fbSQLDatabase: FB_SQLDatabase(sNetID:='', tTimeout:=T#10S);
	fbSQLResult: FB_SQLResult(sNetID:='', tTimeout:=T#10S);
	result: I_TcResultEvent;


	iState: INT;
END_VAR

//Build command


sCmd :='SELECT * FROM [Schedule] ORDER BY [Sequence] ASC';

//State machine
CASE iState OF
0:
//IDLE
fbTON(PT := TIME#4S0MS);
IF fbTON.Q=TRUE THEN
	iState:=1;
	fbTON.IN:=FALSE;
	bError := FALSE; 
ELSE
	fbTON.IN:=TRUE;
END_IF
//Connect
1:
	IF fbSqlDatabase.Connect(1) THEN
		IF fbSqlDatabase.bError THEN
			iState := 255;
			result := fbSqlDatabase.ipTcResultEvent;
			sSeverity := result.Text;
			bError := TRUE; 		
		ELSE
			//If sucessful, point the connection to the sql command function
			fbSqlDatabase.CreateCmd(ADR(fbSqlCommand));
			iState := 2;
		END_IF
	END_IF
2:
//Send the sql command
	IF fbSQLCommand.ExecuteDataReturn(ADR(sCmd), SIZEOF(sCmd), ADR(fbSqlResult)) THEN
		IF fbSQLCommand.bError THEN
			iState := 255;
			result := fbSQLCommand.ipTcResultEvent;
			sSeverity := result.Text;
			bError := TRUE;
		ELSE
			iState := 3; 
			iLines:=fbSqlResult.nDataCount;
		END_IF
	END_IF
		
3:
//Read the sql result
	IF fbSqlResult.Read(0, 1, ADR(arrRecords), SIZEOF(arrRecords), TRUE, TRUE) THEN
		IF fbSqlResult.bError THEN
			result := fbSqlResult.ipTcResultEvent;
			sSeverity := result.Text;
			iState:=255;
			bError := TRUE;
		ELSE 
			iState:=4;
			
			result := fbSqlResult.ipTcResultEvent;
			sSeverity := result.Text;
		END_IF
	

	END_IF
4:
	IF 	fbSqlDatabase.Disconnect() THEN
		bError := FALSE;
		iState:=0;
	END_IF
255:
	IF 	fbSqlDatabase.Disconnect() THEN
		iState:=0;	
		bError := TRUE;
		result := fbSqlResult.ipTcResultEvent;
		sSeverity := result.Text;

	END_IF
	
END_CASE

END_PROGRAM

// ---- POUs/Scheduing/fbGetCurrentProgramName.TcPOU
PROGRAM fbGetCurrentProgramName

VAR_OUTPUT
	arrRecords: ST_ProgramListStruct;
	sSeverity: WSTRING(255);
	bError :BOOL;

	iLines: UDINT;
END_VAR
VAR
	STProgram: ST_ProgramStruct;
	now : TIMESTRUCT;
	nowMinutes : LINT;
	
	previousMinute: LINT;
	
	fbTON: TON := (PT := TIME#10S0MS);

	

	
	fbPLCDBRead : FB_PLCDBRead(sNetID:='',tTimeout:=T#5S);
	fbSqlCommand : FB_SQLCommand(sNetID := '', tTimeout := T#5S);
	
	
	intTime: DINT;
	todTime: TOD;

	sCmd: STRING(255):='SELECT * FROM [Schedule] ORDER BY [Sequence] ASC';

	dIntSqlResult: DINT;
	fbSQLDatabase: FB_SQLDatabase(sNetID:='', tTimeout:=T#10S);
	fbSQLResult: FB_SQLResult(sNetID:='', tTimeout:=T#10S);
	result: I_TcResultEvent;


	iState: INT;
END_VAR

//Build command



sCmd :=CONCAT('SELECT * FROM [ProgramList] WHERE [ID]=',LINT_TO_STRING(GVL.CurrentProgram));

//State machine
CASE iState OF
0:
//IDLE
fbTON(PT := TIME#2S0MS);
IF fbTON.Q=TRUE THEN
	iState:=1;
	fbTON.IN:=FALSE;
	bError := FALSE; 
ELSE
	fbTON.IN:=TRUE;
END_IF
//Connect
1:
	IF fbSqlDatabase.Connect(1) THEN
		IF fbSqlDatabase.bError THEN
			iState := 255;
			result := fbSqlDatabase.ipTcResultEvent;
			sSeverity := result.Text;
			bError := TRUE; 		
		ELSE
			//If sucessful, point the connection to the sql command function
			fbSqlDatabase.CreateCmd(ADR(fbSqlCommand));
			iState := 2;
		END_IF
	END_IF
2:
//Send the sql command
	IF fbSQLCommand.ExecuteDataReturn(ADR(sCmd), SIZEOF(sCmd), ADR(fbSqlResult)) THEN
		IF fbSQLCommand.bError THEN
			iState := 255;
			result := fbSQLCommand.ipTcResultEvent;
			sSeverity := result.Text;
			bError := TRUE;
		ELSE
			iState := 3; 
			iLines:=fbSqlResult.nDataCount;
		END_IF
	END_IF
		
3:
//Read the sql result
	IF fbSqlResult.Read(0, 1, ADR(arrRecords), SIZEOF(arrRecords), TRUE, TRUE) THEN
		IF fbSqlResult.bError THEN
			result := fbSqlResult.ipTcResultEvent;
			sSeverity := result.Text;
			iState:=255;
			bError := TRUE;
		ELSE 
			iState:=4;
			
			result := fbSqlResult.ipTcResultEvent;
			sSeverity := result.Text;
		END_IF
	

	END_IF
4:
	IF 	fbSqlDatabase.Disconnect() THEN
		bError := FALSE;
		iState:=0;
	END_IF
255:
	IF 	fbSqlDatabase.Disconnect() THEN
		iState:=0;	
		bError := TRUE;
		result := fbSqlResult.ipTcResultEvent;
		sSeverity := result.Text;

	END_IF
	
END_CASE

END_PROGRAM

// ---- POUs/DeleteOldData.TcPOU
		PROGRAM DeleteOldData

VAR_OUTPUT
	arrRecords: ST_ProgramListStruct;
	sSeverity: WSTRING(255);
	bError :BOOL;

	iLines: UDINT;
END_VAR
VAR
	STProgram: ST_ProgramStruct;
	nowMinutes : LINT;
	
	previousMinute: LINT;
	
	fbTON: TON := (PT := TIME#10S0MS);

	

	
	fbPLCDBRead : FB_PLCDBRead(sNetID:='',tTimeout:=T#5S);
	fbSqlCommand : FB_SQLCommand(sNetID := '', tTimeout := T#5S);
	
	
	intTime: DINT;
	todTime: TOD;

	sCmd: STRING(255):='SELECT * FROM [Schedule] ORDER BY [Sequence] ASC';

	dIntSqlResult: DINT;
	fbSQLDatabase: FB_SQLDatabase(sNetID:='', tTimeout:=T#10S);
	fbSQLResult: FB_SQLResult(sNetID:='', tTimeout:=T#10S);
	result: I_TcResultEvent;


	iState: INT;
	ulNow: ULINT;
	
	TwoYearsAgo: LTIME := LTIME#1051200m0s0ms0us0ns;
	dtNow: DATE_AND_TIME;
END_VAR

//Build command
sCmd :='DELETE FROM Logger WHERE Timestamp <= datetime("now","-2 year")';

//State machine
CASE iState OF
0:
//IDLE
fbTON(PT := TIME#900S0MS);
IF fbTON.Q=TRUE THEN
	iState:=1;
	fbTON.IN:=FALSE;
	bError := FALSE; 
ELSE
	fbTON.IN:=TRUE;
END_IF
//Connect
1:
	IF fbSqlDatabase.Connect(1) THEN
		IF fbSqlDatabase.bError THEN
			iState := 255;
			result := fbSqlDatabase.ipTcResultEvent;
			sSeverity := result.Text;
			bError := TRUE; 		
		ELSE
			//If sucessful, point the connection to the sql command function
			fbSqlDatabase.CreateCmd(ADR(fbSqlCommand));
			iState := 2;
		END_IF
	END_IF
2:
//Send the sql command
	IF fbSQLCommand.ExecuteDataReturn(ADR(sCmd), SIZEOF(sCmd), ADR(fbSqlResult)) THEN
		IF fbSQLCommand.bError THEN
			iState := 255;
			result := fbSQLCommand.ipTcResultEvent;
			sSeverity := result.Text;
			bError := TRUE;
		ELSE
			iState := 3; 
			iLines:=fbSqlResult.nDataCount;
		END_IF
	END_IF
		
3:
//Read the sql result
	IF fbSqlResult.Read(0, 1, ADR(arrRecords), SIZEOF(arrRecords), TRUE, TRUE) THEN
		IF fbSqlResult.bError THEN
			result := fbSqlResult.ipTcResultEvent;
			sSeverity := result.Text;
			iState:=255;
			bError := TRUE;
		ELSE 
			iState:=4;
			result := fbSqlResult.ipTcResultEvent;
			sSeverity := result.Text;
		END_IF
	END_IF
4:
	IF 	fbSqlDatabase.Disconnect() THEN
		bError := FALSE;
		iState:=0;
	END_IF
255:
	IF 	fbSqlDatabase.Disconnect() THEN
		iState:=0;	
		bError := TRUE;
		result := fbSqlResult.ipTcResultEvent;
		sSeverity := result.Text;

	END_IF
	
END_CASE

END_PROGRAM

// ---- POUs/Program Setpoints/DatabaseStateMachine.TcPOU
PROGRAM DatabaseStateMachine
VAR_INPUT
	
	bStepStart: BOOL:=TRUE;

END_VAR
	
VAR_OUTPUT
	allOutputsSet:BOOL;
END_VAR

VAR
	iState: INT;
	nextLine:ST_ProgramStruct;
	previousLine:ST_ProgramStruct;
	fbTON: TON := (PT := TIME#10S0MS);
	fbScaleValue: scaleValue;
	TempModeSwitchTrigger: F_TRIG;
		
	errorText: WSTRING(255);
	bError: BOOL;
	bSuccess: BOOL;
	iLines: UDINT;
	
	
	CalculateTemp: fbCalculateSetpoint;
	CalculateLight1: fbCalculateSetpoint;
	CalculateLight2: fbCalculateSetpoint;
	CalculateHumidity: fbCalculateSetpoint;
	CalculateDO10: fbCalculateSetpoint;
	CalculateDO11: fbCalculateSetpoint;
	
	
	
	nextLineTemp: ST_ProgramStruct;
	previousLineTemp: ST_ProgramStruct;
	
	nextLineLight1: ST_ProgramStruct;
	previousLineLight1: ST_ProgramStruct;
	
	nextLineLight2: ST_ProgramStruct;
	previousLineLight2: ST_ProgramStruct;
	
	nextLineHumidity: ST_ProgramStruct;
	previousLineHumidity: ST_ProgramStruct;
	
	nextLineDO10: ST_ProgramStruct;
	previousLineDO10: ST_ProgramStruct;
	
	nextLineDO11: ST_ProgramStruct;
	previousLineDO11: ST_ProgramStruct;
	
	//temp holder for conversion to bool
	tempVar:REAL;
	
END_VAR

//In the case that the user switches from step mode to ramp mode, we need to set the current setpoint to the current value
//Really only needed for analog values controlled by a PID
//Like temperature, humidity...maybe CO2?

TempModeSwitchTrigger(CLK:=GVL.TempStepmode);

IF TempModeSwitchTrigger.Q THEN
	GVL.TempSetpoint:=GVL.Temp;
END_IF



CASE iState OF
	
	//Check connection
	0:
		
		fbTON(PT := TIME#1S0MS);
		allOutputsSet:=FALSE;
		IF fbTON.Q=TRUE THEN
			DBConnector();
			IF DBConnector.fbSQLDatabase.bConnected THEN
				iState:=iState+1;
				fbTON.IN:=FALSE;
			END_IF
		ELSE
			fbTON.IN:=TRUE;
		END_IF
		
		
	
	1:
		//GET TEMPERATURE
		QueryProgram(sColumn:='[Temperature]');
		IF QueryProgram.bSuccess THEN
			iState:=iState+1;
			nextLineTemp:=QueryProgram.arrRecords;
			previousLineTemp:=QueryProgram.previousLine;
			
			IF QueryProgram.bEndOfProgram THEN
				nextLineTemp.iTime:=nextLineTemp.iTime+1440;
			END_IF
			
			IF bStepStart=TRUE THEN
				GVL.TempSetpoint:=GVL.Temp;
			END_IF
			
		END_IF
		
		

	
		
	2:
		//GET LIGHT 1 LEVEL
		QueryProgram(sColumn:='[Light1_MH]');
		
		IF QueryProgram.bSuccess THEN
				iState:=iState+1;
				nextLineLight1:=QueryProgram.arrRecords;
				previousLineLight1:=QueryProgram.previousLine;
				
				IF QueryProgram.bEndOfProgram THEN
					nextLineLight1.iTime:=nextLineLight1.iTime+1440;
				END_IF
				
		END_IF
	3:
		//GET LIGHT 2 LEVEL
		QueryProgram(sColumn:='[Light2_HPS]');
		
		IF QueryProgram.bSuccess THEN
				iState:=iState+1;
				nextLineLight2:=QueryProgram.arrRecords;
				previousLineLight2:=QueryProgram.previousLine;
				
				IF QueryProgram.bEndOfProgram THEN
					nextLineLight2.iTime:=nextLineLight2.iTime+1440;
				END_IF
				
		END_IF
	4:
		//GET HUMIDITY
		QueryProgram(sColumn:='[Humidity]');
		
		IF QueryProgram.bSuccess THEN
				iState:=iState+1;
				nextLineHumidity:=QueryProgram.arrRecords;
				previousLineHumidity:=QueryProgram.previousLine;
				
				IF QueryProgram.bEndOfProgram THEN
					nextLineHumidity.iTime:=nextLineHumidity.iTime+1440;
				END_IF
				
		END_IF
	5:
		//DIGITAL OUT 10
		QueryProgram(sColumn:='[DigitalOut10]');
		
		IF QueryProgram.bSuccess THEN
				iState:=iState+1;
				nextLineDO10:=QueryProgram.arrRecords;
				previousLineDO10:=QueryProgram.previousLine;
				
				IF QueryProgram.bEndOfProgram THEN
					nextLineDO10.iTime:=nextLineLight2.iTime+1440;
				END_IF
				
		END_IF
	6:
		//DIGITAL OUT 11
		QueryProgram(sColumn:='[DigitalOut11]');
		
		IF QueryProgram.bSuccess THEN
				iState:=iState+1;
				nextLineDO11:=QueryProgram.arrRecords;
				previousLineDO11:=QueryProgram.previousLine;
				
				IF QueryProgram.bEndOfProgram THEN
					nextLineDO11.iTime:=nextLineLight2.iTime+1440;
				END_IF
				
		END_IF
	
		
	7:
	//Success!
	allOutputsSet:=TRUE;
	iState:=0;
		

END_CASE


//Using the setpoints we just got above,
//Calculate what the target setpoint is based on
//If we're in ramp mode, step mode, what time it is, etc
CalculateTemp(
	currentValue:=GVL.Temp,
	nextSetpointValue:= nextLineTemp.Temperature, 
	nextSetpointTime:= nextLineTemp.iTime, 
	currentSetpoint:= GVL.TempSetpoint,
	previousSetpoint:=previousLineTemp.Temperature,
	previousSetpointTime:=previousLineTemp.iTime,
	stepMode:= GVL.TempStepmode, 
	setpoint=> GVL.TempSetpoint,
	bStepStart:=FALSE,
	);
	
	
CalculateLight1(
		currentValue:=GVL.Light1Percent,
		nextSetpointValue:= nextLineLight1.Light1, 
		nextSetpointTime:= nextLineLight1.iTime, 
		currentSetpoint:= GVL.Light1Percent,
		previousSetpoint:=previousLineLight1.Light1,
		previousSetpointTime:=previousLineLight1.iTime, 
		stepMode:= GVL.Light1Stepmode, 
		setpoint=> GVL.Light1Percent,
		bStepStart:=bStepStart);
		
fbScaleValue(rInputPercent:=GVL.Light1Percent,rMaxValue:=GVL.Light1Max,iScaled=>GVL.Light1Level);

CalculateLight2(
		currentValue:=GVL.Light2Percent,
		nextSetpointValue:= nextLineLight2.Light2, 
		nextSetpointTime:= nextLineLight2.iTime, 
		currentSetpoint:= GVL.Light2Percent,
		previousSetpoint:=previousLineLight2.Light2,
		previousSetpointTime:=previousLineLight2.iTime, 
		stepMode:= GVL.Light2Stepmode, 
		setpoint=> GVL.Light2Percent,
		bStepStart:=bStepStart);
		
fbScaleValue(rInputPercent:=GVL.Light2Percent,rMaxValue:=GVL.Light2Max,iScaled=>GVL.Light2Level);

CalculateHumidity(
		currentValue:=GVL.Humidity,
		nextSetpointValue:= nextLineHumidity.humidity, 
		nextSetpointTime:= nextLineHumidity.iTime, 
		currentSetpoint:= GVL.HumiditySetpoint,
		previousSetpoint:=previousLineHumidity.humidity,
		previousSetpointTime:=previousLineHumidity.iTime, 
		stepMode:= GVL.HumidityStepmode, 
		setpoint=> GVL.HumiditySetpoint,
		bStepStart:=bStepStart);

	
CalculateDO10(
		currentValue:=BOOL_TO_REAL(IO_VARS.AUX2),
		nextSetpointValue:= BOOL_TO_REAL(nextLineDO10.DO10), 
		nextSetpointTime:= nextLineDO10.iTime, 
		currentSetpoint:= BOOL_TO_REAL(IO_VARS.AUX2),
		previousSetpoint:=BOOL_TO_REAL(previousLineDO10.DO10),
		previousSetpointTime:=previousLineDO10.iTime, 
		stepMode:= TRUE,//Digital Auxillaries are always step mode 
		setpoint=> tempVar,
		bStepStart:=bStepStart);
		
IO_VARS.AUX2:=REAL_TO_BOOL(tempVar);
		
CalculateDO11(
		currentValue:=BOOL_TO_REAL(IO_VARS.AUX3),
		nextSetpointValue:= BOOL_TO_REAL(nextLineDO11.DO11), 
		nextSetpointTime:= nextLineDO11.iTime, 
		currentSetpoint:= BOOL_TO_REAL(IO_VARS.AUX3),
		previousSetpoint:=BOOL_TO_REAL(previousLineDO11.DO11),
		previousSetpointTime:=previousLineDO11.iTime, 
		stepMode:= TRUE,//Digital Auxillaries are always step mode 
		setpoint=> tempVar,
		bStepStart:=bStepStart);
		
IO_VARS.AUX3:=REAL_TO_BOOL(tempVar);

END_PROGRAM

// ---- FB/scaleValue.TcPOU
FUNCTION_BLOCK scaleValue
VAR_INPUT
	rInputPercent:REAL;
	rMaxValue:REAL;

END_VAR
VAR_OUTPUT
	
	iScaled:INT;
END_VAR
VAR
END_VAR

iScaled:=REAL_TO_INT(rInputPercent*rMaxValue/100);

END_FUNCTION_BLOCK

// ---- FB/fbCalculateSetpoint.TcPOU
FUNCTION_BLOCK fbCalculateSetpoint
VAR_INPUT
	currentValue:REAL;
	nextSetpointValue:REAL;
	nextSetpointTime:LINT;
	currentSetpoint:REAL;
	previousSetpoint:REAL;
	previousSetpointTime:LINT;
	stepMode:BOOL;
	rampingMultiplier:REAL;
	bStepStart:BOOL;
END_VAR
VAR_OUTPUT
	setpoint:REAL;
	
END_VAR
VAR
	
	NextTemp: LREAL;
	
	nowMinutes: LINT;
	nowSeconds:LINT;
	now: TIMESTRUCT;
	fbTON: TON := (PT := TIME#1s0ms);
	
END_VAR


now := GVL.fbLocalSystemTime.systemTime;
nowMinutes := now.wHour*60+now.wMinute;
nowSeconds :=nowMinutes*60+now.wSecond;


fbTON();



IF stepMode=TRUE THEN
	
	IF nowMinutes >= nextSetpointTime THEN
		setpoint := nextSetpointValue;
	ELSE
		setpoint:=previousSetpoint;
	END_IF
	
ELSE

	//Ramp
	IF bStepStart THEN
	
		IF (nextSetpointTime-previousSetpointTime)<>0 THEN
			setpoint:= ((nextSetpointValue - previousSetpoint)/((nextSetpointTime-previousSetpointTime)))*(nowMinutes-previousSetpointTime)+previousSetpoint;
		END_IF
	
	ELSE
		IF ((nextSetpointTime*60)-nowSeconds)<>0 THEN
			setpoint:= ((nextSetpointValue - currentSetpoint)/(((nextSetpointTime*60)-nowSeconds)))*(GVL.cycleTime)+currentSetpoint;
		ELSIF ((nextSetpointTime*60)-nowSeconds)=0 THEN
			setpoint:=nextSetpointValue;
		END_IF
	END_IF
	
END_IF

END_FUNCTION_BLOCK

// ---- POUs/Program Setpoints/DBConnector.TcPOU
PROGRAM DBConnector


VAR_OUTPUT

	sSeverity: WSTRING(255);
	bError :BOOL;

END_VAR
VAR

	fbSQLDatabase: FB_SQLDatabase(sNetID:='', tTimeout:=T#10S);
	result: I_TcResultEvent;
	iState: INT;
END_VAR


//State machine
CASE iState OF

//Connect
0:
	IF fbSqlDatabase.Connect(1) THEN
		IF fbSqlDatabase.bError THEN
			iState := 255;
			result := fbSqlDatabase.ipTcResultEvent;
			sSeverity := result.Text;
			bError := TRUE; 		
		ELSE
			iState := 1;
		END_IF
	END_IF
1:
//Make sure it's still connected
	IF fbSqlDatabase.bConnected THEN
		result := fbSqlDatabase.ipTcResultEvent;
		sSeverity := result.Text;
		bError := fbSqlDatabase.bError;		
	ELSE
		iState := 255;
		result := fbSqlDatabase.ipTcResultEvent;
		sSeverity := result.Text;
		bError := fbSqlDatabase.bError;
	END_IF

255:
//Error handling
	//ADSLOGSTR(msgCtrlMask := ADSLOG_MSGTYPE_ERROR OR ADSLOG_MSGTYPE_MSGBOX, msgFmtStr := 'Oh what have you done? %s', strArg := WSTRING_TO_STRING(result.Text));
	IF fbSqlDatabase.Disconnect() THEN
			
			iState := 0;
			result := fbSqlDatabase.ipTcResultEvent;
			sSeverity := result.Text;
			bError := fbSqlDatabase.bError;
	
	END_IF
 	
END_CASE

END_PROGRAM

// ---- POUs/Program Setpoints/QueryProgram.TcPOU
PROGRAM QueryProgram
VAR_INPUT
	sColumn:STRING(255);
END_VAR
VAR_OUTPUT
	arrRecords: ST_ProgramStruct;
	previousLine:ST_ProgramStruct;
	sSeverity: WSTRING(255);
	bError :BOOL;
	bEndOfProgram:BOOL;
	iLines: UDINT;
	bSuccess: BOOL;
	
	
END_VAR
VAR
	STProgram: ST_ProgramStruct;
	now : TIMESTRUCT;
	nowMinutes : LINT;
	fbTON: TON := ();
	fbSQLDatabase: FB_SQLDatabase(sNetID:='', tTimeout:=T#10S);
	fbPLCDBRead : FB_PLCDBRead(sNetID:='',tTimeout:=T#5S);
	fbSqlCommand : FB_SQLCommand(sNetID := '', tTimeout := T#5S);
	
	
	intTime: DINT;
	todTime: TOD;

	sCmd: STRING(255);

	dIntSqlResult: DINT;
	
	fbSQLResult: FB_SQLResult(sNetID:='', tTimeout:=T#10S);
	result: I_TcResultEvent;


	iState: INT;
	
	
	iPreviousLines: UDINT;
END_VAR




now := GVL.fbLocalSystemTime.systemTime;
nowMinutes := now.wHour*60+now.wMinute;
fbSQLDatabase:=DBConnector.fbSQLDatabase;

//State machine
CASE iState OF
0:
//IDLE
fbTON(PT := TIME#250MS);
bSuccess:=FALSE;
bEndOfProgram:=FALSE;
//Build command

sCmd :=CONCAT('SELECT * FROM [Programs] WHERE [ProgramNameID]=',LINT_TO_STRING(GVL.CurrentProgram));
sCmd :=CONCAT(sCmd,' AND [time]>');
sCmd := CONCAT(sCMD,LINT_TO_STRING(nowMinutes));
sCmd :=CONCAT(sCmd,' AND ');
sCmd := CONCAT(sCMD,sColumn);
sCmd := CONCAT(sCMD,' IS NOT NULL');
sCmd:= CONCAT(sCMD,' ORDER BY [time] ASC');
 
IF fbTON.Q=TRUE THEN
	iState:=1;
	fbTON.IN:=FALSE;
	bError := FALSE;
	
ELSE
	fbTON.IN:=TRUE;
END_IF
//Connect
1:

		IF fbSqlDatabase.bError THEN
			iState := 255;
			result := fbSqlDatabase.ipTcResultEvent;
			sSeverity := result.Text;
			 		
		ELSE
			//If sucessful, point the connection to the sql command function
			fbSqlDatabase.CreateCmd(ADR(fbSqlCommand));
			iState := 2;
		END_IF

2:
//Send the sql command
	IF fbSQLCommand.ExecuteDataReturn(ADR(sCmd), SIZEOF(sCmd), ADR(fbSqlResult)) THEN
		IF fbSQLCommand.bError THEN
			iState := 255;
			result := fbSQLCommand.ipTcResultEvent;
			sSeverity := result.Text;
			bError := TRUE;
		ELSE
			iState := 3;
			iLines:=fbSqlResult.nDataCount; 
		END_IF
	END_IF
		
3:
//Read the sql result
//If there are more than 0 lines, we're good
//If there are 0 lines we have reached the end of the program and we need to query tomorrow's program

IF iLines>0 THEN
	
	IF fbSqlResult.Read(0, 1, ADR(arrRecords), SIZEOF(arrRecords), TRUE, TRUE) THEN
		IF fbSqlResult.bError THEN
			result := fbSqlResult.ipTcResultEvent;
			sSeverity := result.Text;
			iState:=255;
			bError := TRUE;
		ELSE 
			iState:=4;
			
			result := fbSqlResult.ipTcResultEvent;
			sSeverity := result.Text;
		END_IF
	

	END_IF
	
ELSE

bEndOfProgram:=TRUE;
sCmd :=CONCAT('SELECT  *  FROM [Programs]  WHERE [ProgramNameID]=',LINT_TO_STRING(GVL.NextProgram));
sCmd :=CONCAT(sCmd,' AND ');
sCmd := CONCAT(sCMD,sColumn);
sCmd := CONCAT(sCMD,' IS NOT NULL');
sCmd := CONCAT(sCMD,' ORDER BY [time] ASC');
//Go back to state 2 and redo the query
iState:=2;

END_IF
4:
//Now build a command and query the PREVIOUS line in the program
sCmd := CONCAT('SELECT  *  FROM [Programs]  WHERE [ProgramNameID]=',LINT_TO_STRING(GVL.CurrentProgram));
sCmd := CONCAT(sCmd,' AND [time] <=');
sCmd := CONCAT(sCMD,LINT_TO_STRING(nowMinutes));
sCmd := CONCAT(sCmd,' AND ');
sCmd := CONCAT(sCMD,sColumn);
sCmd := CONCAT(sCMD,' IS NOT NULL');
sCmd := CONCAT(sCMD,' ORDER BY [time] DESC');	
	IF fbSQLCommand.ExecuteDataReturn(ADR(sCmd), SIZEOF(sCmd), ADR(fbSqlResult)) THEN
		IF fbSQLCommand.bError THEN
			iState := 255;
			result := fbSQLCommand.ipTcResultEvent;
			sSeverity := result.Text;
			bError := TRUE;
		ELSE
			iState := 5; 
			iPreviousLines:=fbSqlResult.nDataCount;
		END_IF
	END_IF

5:
//read the previous line
//If there IS a previous line then
IF iPreviousLines>0 THEN
 
	IF fbSqlResult.Read(0, 1, ADR(previousLine), SIZEOF(previousLine), TRUE, TRUE) THEN
		IF fbSqlResult.bError THEN
			result := fbSqlResult.ipTcResultEvent;
			sSeverity := result.Text;
			iState:=255;
			bError := TRUE;
		ELSE 
			//We're done go back to the beginning
			iState:=0;
			bSuccess:=TRUE; 
			result := fbSqlResult.ipTcResultEvent;
			sSeverity := result.Text;
			
		END_IF
	

	END_IF
	
//If there is NO previous line...the previous line is the next line
ELSE
	previousLine:=arrRecords;
	//We're done go back to the beginning
	iState:=0;
	bSuccess:=TRUE; 
	result := fbSqlResult.ipTcResultEvent;
	sSeverity := result.Text;
END_IF


255:
	//Record the error....I need to change this to actually record the errors
		ADSLOGSTR(msgCtrlMask := ADSLOG_MSGTYPE_ERROR OR ADSLOG_MSGTYPE_MSGBOX, msgFmtStr := 'Oh god what have you done? %s', strArg := WSTRING_TO_STRING(result.Text));
		iState:=0;	
		bError := TRUE;
		result := fbSqlResult.ipTcResultEvent;
		sSeverity := result.Text;
	

END_CASE

END_PROGRAM

// ---- POUs/OLD NOT USED/POU.TcPOU
PROGRAM POU
VAR
	error: UINT;
	TempPID: FB_BasicPID;
	test: BOOL;

END_VAR

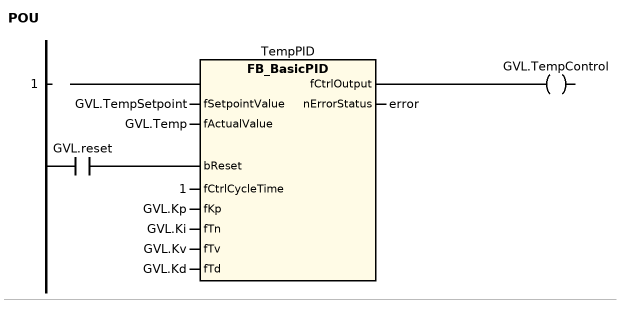
// NETWORK 1
TempPID(
    fSetpointValue := GVL.TempSetpoint,
    fActualValue := GVL.Temp,
    bReset := GVL.reset,
    fCtrlCycleTime := 1,
    fKp := GVL.Kp,
    fTn := GVL.Ki,
    fTv := GVL.Kv,
    fTd := GVL.Kd,
    nErrorStatus => error); // FB_BasicPID
GVL.TempControl := TempPID.fCtrlOutput;

END_PROGRAM

// ---- POUs/OLD NOT USED/fbGetNextLine.TcPOU
PROGRAM fbGetNextLine

VAR_OUTPUT
	arrRecords: ST_ProgramStruct;
	sSeverity: WSTRING(255);
	bError :BOOL;
	iLines: UDINT;
END_VAR
VAR
	STProgram: ST_ProgramStruct;
	now : TIMESTRUCT;
	nowMinutes : LINT;
	fbTON: TON := (PT := TIME#10S0MS);

	fbPLCDBRead : FB_PLCDBRead(sNetID:='',tTimeout:=T#5S);
	fbSqlCommand : FB_SQLCommand(sNetID := '', tTimeout := T#5S);
	
	
	intTime: DINT;
	todTime: TOD;

	sCmd: STRING(255);

	dIntSqlResult: DINT;
	fbSQLDatabase: FB_SQLDatabase(sNetID:='', tTimeout:=T#10S);
	fbSQLResult: FB_SQLResult(sNetID:='', tTimeout:=T#10S);
	result: I_TcResultEvent;


	iState: INT;
END_VAR

//Build command


now := GVL.fbLocalSystemTime.systemTime;
nowMinutes := now.wHour*60+now.wMinute;


sCmd :=CONCAT('SELECT * FROM [Programs] WHERE [ProgramNameID]=',LINT_TO_STRING(GVL.CurrentProgram));

sCmd :=CONCAT(sCmd,' AND [time]>');

sCmd := CONCAT(sCMD,LINT_TO_STRING(nowMinutes));

sCmd:= CONCAT(sCMD,' ORDER BY [time] ASC');
//State machine
CASE iState OF
0:
//IDLE
fbTON();
IF fbTON.Q=TRUE THEN
	iState:=1;
	fbTON.IN:=FALSE;
	bError := FALSE; 
ELSE
	fbTON.IN:=TRUE;
END_IF
//Connect
1:
	IF fbSqlDatabase.Connect(1) THEN
		IF fbSqlDatabase.bError THEN
			iState := 255;
			result := fbSqlDatabase.ipTcResultEvent;
			sSeverity := result.Text;
			bError := TRUE; 		
		ELSE
			//If sucessful, point the connection to the sql command function
			fbSqlDatabase.CreateCmd(ADR(fbSqlCommand));
			iState := 2;
		END_IF
	END_IF
2:
//Send the sql command
	IF fbSQLCommand.ExecuteDataReturn(ADR(sCmd), SIZEOF(sCmd), ADR(fbSqlResult)) THEN
		IF fbSQLCommand.bError THEN
			iState := 255;
			result := fbSQLCommand.ipTcResultEvent;
			sSeverity := result.Text;
			bError := TRUE;
		ELSE
			iState := 3;
			iLines:=fbSqlResult.nDataCount; 
		END_IF
	END_IF
		
3:
//Read the sql result
	
	IF fbSqlResult.Read(0, 1, ADR(arrRecords), SIZEOF(arrRecords), TRUE, TRUE) THEN
		IF fbSqlResult.bError THEN
			result := fbSqlResult.ipTcResultEvent;
			sSeverity := result.Text;
			iState:=255;
			bError := TRUE;
		ELSE 
			iState:=4;
			
			result := fbSqlResult.ipTcResultEvent;
			sSeverity := result.Text;
		END_IF
	

	END_IF
4:
//Disconnect
	IF 	fbSqlDatabase.Disconnect() THEN
		IF fbSqlDatabase.bError THEN
        	iState := 255;
		ELSE
			iState := 0;
			bError := FALSE;
		END_IF

	END_IF
255:
//Record the error....I need to change this to actually record the errors
		iState:=0;	
		bError := TRUE;
		result := fbSqlResult.ipTcResultEvent;
		sSeverity := result.Text;
		fbSqlDatabase.Disconnect();

END_CASE

END_PROGRAM

// ---- POUs/OLD NOT USED/fbGetNextLineAfterMidnight.TcPOU
PROGRAM fbGetNextLineAfterMidnight

VAR_OUTPUT
	arrRecords: ST_ProgramStruct;
	sSeverity: WSTRING(255);
	bError :BOOL;

	iLines: UDINT;
END_VAR
VAR
	STProgram: ST_ProgramStruct;
	now : TIMESTRUCT;
	nowMinutes : LINT;
	
	previousMinute: LINT;
	
	fbTON: TON := (PT := TIME#10S0MS);

	

	
	fbPLCDBRead : FB_PLCDBRead(sNetID:='',tTimeout:=T#5S);
	fbSqlCommand : FB_SQLCommand(sNetID := '', tTimeout := T#5S);
	
	
	intTime: DINT;
	todTime: TOD;

	sCmd: STRING(255);

	dIntSqlResult: DINT;
	fbSQLDatabase: FB_SQLDatabase(sNetID:='', tTimeout:=T#10S);
	fbSQLResult: FB_SQLResult(sNetID:='', tTimeout:=T#10S);
	result: I_TcResultEvent;


	iState: INT;
END_VAR

//Build command


now := GVL.fbLocalSystemTime.systemTime;
nowMinutes := now.wHour*60+now.wMinute;



sCmd :=CONCAT('SELECT  *  FROM [Programs]  WHERE [ProgramNameID]=',LINT_TO_STRING(GVL.NextProgram));

sCmd:= CONCAT(sCMD,' ORDER BY [time] ASC');

//State machine
CASE iState OF
0:
//IDLE
fbTON();
IF fbTON.Q=TRUE THEN
	iState:=1;
	fbTON.IN:=FALSE;
	bError := FALSE; 
ELSE
	fbTON.IN:=TRUE;
END_IF
//Connect
1:
	IF fbSqlDatabase.Connect(1) THEN
		IF fbSqlDatabase.bError THEN
			iState := 255;
			result := fbSqlDatabase.ipTcResultEvent;
			sSeverity := result.Text;
			bError := TRUE; 		
		ELSE
			//If sucessful, point the connection to the sql command function
			fbSqlDatabase.CreateCmd(ADR(fbSqlCommand));
			iState := 2;
		END_IF
	END_IF
2:
//Send the sql command
	IF fbSQLCommand.ExecuteDataReturn(ADR(sCmd), SIZEOF(sCmd), ADR(fbSqlResult)) THEN
		IF fbSQLCommand.bError THEN
			iState := 255;
			result := fbSQLCommand.ipTcResultEvent;
			sSeverity := result.Text;
			bError := TRUE;
		ELSE
			iState := 3; 
			iLines:=fbSqlResult.nDataCount;
		END_IF
	END_IF
		
3:
//Read the sql result
	IF fbSqlResult.Read(0, 1, ADR(arrRecords), SIZEOF(arrRecords), TRUE, TRUE) THEN
		IF fbSqlResult.bError THEN
			result := fbSqlResult.ipTcResultEvent;
			sSeverity := result.Text;
			iState:=255;
			bError := TRUE;
		ELSE 
			iState:=4;
			
			result := fbSqlResult.ipTcResultEvent;
			sSeverity := result.Text;
		END_IF
	

	END_IF
4:
	IF 	fbSqlDatabase.Disconnect() THEN
		bError := FALSE;
		iState:=0;
	END_IF
255:
	IF 	fbSqlDatabase.Disconnect() THEN
		iState:=0;	
		bError := TRUE;
		result := fbSqlResult.ipTcResultEvent;
		sSeverity := result.Text;

	END_IF
	
END_CASE

END_PROGRAM

// ---- POUs/OLD NOT USED/GetPreviousLine.TcPOU
PROGRAM GetPreviousLine

VAR_OUTPUT
	arrRecords: ST_ProgramStruct;
	sSeverity: WSTRING(255);
	bError :BOOL;

	iLines: UDINT;
END_VAR
VAR
	STProgram: ST_ProgramStruct;
	now : TIMESTRUCT;
	nowMinutes : LINT;
	
	previousMinute: LINT;

	

	
	fbPLCDBRead : FB_PLCDBRead(sNetID:='',tTimeout:=T#5S);
	fbSqlCommand : FB_SQLCommand(sNetID := '', tTimeout := T#5S);
	
	
	intTime: DINT;
	todTime: TOD;

	sCmd: STRING(255);

	dIntSqlResult: DINT;
	fbSQLDatabase: FB_SQLDatabase(sNetID:='', tTimeout:=T#10S);
	fbSQLResult: FB_SQLResult(sNetID:='', tTimeout:=T#10S);
	result: I_TcResultEvent;


	iState: INT;
	fbTON: TON := (PT := TIME#10s0ms);

END_VAR

//Build command


now := GVL.fbLocalSystemTime.systemTime;
nowMinutes := now.wHour*60+now.wMinute;



sCmd :=CONCAT('SELECT  *  FROM [Programs]  WHERE [ProgramNameID]=',LINT_TO_STRING(GVL.CurrentProgram));

sCmd :=CONCAT(sCmd,' AND [time] <=');

sCmd := CONCAT(sCMD,LINT_TO_STRING(nowMinutes));

sCmd:= CONCAT(sCMD,' ORDER BY [time] DESC');
//State machine
CASE iState OF
0:
//IDLE
fbTON();
IF fbTON.Q=TRUE THEN
	iState:=1;
	fbTON.IN:=FALSE;
	bError := FALSE; 
ELSE
	fbTON.IN:=TRUE;
END_IF
//Connect
1:
	IF fbSqlDatabase.Connect(1) THEN
		IF fbSqlDatabase.bError THEN
			iState := 255;
			result := fbSqlDatabase.ipTcResultEvent;
			sSeverity := result.Text;
			bError := TRUE; 		
		ELSE
			//If sucessful, point the connection to the sql command function
			fbSqlDatabase.CreateCmd(ADR(fbSqlCommand));
			iState := 2;
		END_IF
	END_IF
2:
//Send the sql command
	IF fbSQLCommand.ExecuteDataReturn(ADR(sCmd), SIZEOF(sCmd), ADR(fbSqlResult)) THEN
		IF fbSQLCommand.bError THEN
			iState := 255;
			result := fbSQLCommand.ipTcResultEvent;
			sSeverity := result.Text;
			bError := TRUE;
		ELSE
			iState := 3; 
			iLines:=fbSqlResult.nDataCount;
		END_IF
	END_IF
		
3:
//Read the sql result
	IF fbSqlResult.Read(0, 1, ADR(arrRecords), SIZEOF(arrRecords), TRUE, TRUE) THEN
		IF fbSqlResult.bError THEN
			result := fbSqlResult.ipTcResultEvent;
			sSeverity := result.Text;
			iState:=255;
			bError := TRUE;
		ELSE 
			iState:=4;
			
			result := fbSqlResult.ipTcResultEvent;
			sSeverity := result.Text;
		END_IF
	

	END_IF
4:
	IF 	fbSqlDatabase.Disconnect() THEN
		bError := FALSE;
		iState:=0;
	END_IF
255:
	IF 	fbSqlDatabase.Disconnect() THEN
		iState:=0;	
		bError := TRUE;
		result := fbSqlResult.ipTcResultEvent;
		sSeverity := result.Text;
	END_IF
	
END_CASE

END_PROGRAM

// ---- GlobalTextList.TcGTLO
TEXTLIST GlobalTextList
  746 = '%.0f'
  406 = '%.1f'
  576 = '%.1f%%'
  940 = '%.3f'
  386 = '%2.0f'
  388 = '%2.0f %%'
  166 = '%2.0f%%'
  1002 = '%2.1f C'
  383 = '%2.2f'
  975 = '%2.2f C'
  489 = '%2.2f g/m³'
  987 = '%d'
  947 = '%i'
  195 = '%s'
  477 = '%X'
  748 = 'Abs. Humidity'
  243 = 'Acknowledge Alarms'
  599 = 'Admin'
  134 = 'Alarm'
  405 = 'Alarm Note'
  194 = 'Alarms'
  742 = 'Contactor'
  745 = 'Cooling                         Heating'
  945 = 'Cooling PID'
  747 = 'Current Program'
  398 = 'Current Program:'
  404 = 'Date & Time'
  162 = 'DO 10'
  741 = 'DO 11'
  409 = 'DO 9'
  656 = 'Enable'
  948 = 'Fan Speed %'
  581 = 'For this many seconds:'
  82 = 'Friday'
  191 = 'Graph'
  853 = 'Heaters'
  949 = 'Heating PID'
  241 = 'High Temperature Limit'
  189 = 'Home'
  61 = 'Hour'
  298 = 'HPS'
  496 = 'HPS Lvl 1'
  850 = 'HPS Lvl 2'
  851 = 'HPS Lvl 3'
  481 = 'Hum. Calibration Alarm'
  297 = 'Humidity'
  852 = 'Humidity Add'
  296 = 'Humidity PID'
  507 = 'Humidity sensor 1'
  762 = 'Humidity sensor 2'
  442 = 'Humidity sensor Humidity sensor 1'
  68 = 'Humidity Valve'
  1017 = 'If the percent difference between\n the two sensors is greater than \nthese values, the system will alarm\n and stop.'
  396 = 'If the percent difference between\nthe two sensors is greater than \nthese values, the system will alarm\nand stop.'
  79 = 'If the percent difference between the two sensors is greater than these values, the system will alarm and stop.'
  244 = 'In ramp mode, this is the deviation from \nthe setpoint\n\nIn step mode, these are absolute values'
  193 = 'IO'
  941 = 'Kp'
  657 = 'Level 1 Light'
  74 = 'Level 1 Light 1'
  548 = 'Level 1 Light 2'
  658 = 'Level 2 Light'
  40 = 'Level 2 Light 1'
  376 = 'Level 2 Light 2'
  709 = 'Level 3 Light 1'
  369 = 'Level 3 Light 2'
  743 = 'Light Level 1'
  744 = 'Light Level 2'
  196 = 'Log In'
  199 = 'Log Out'
  242 = 'Low Temperature Limit'
  192 = 'Manual Mode'
  655 = 'Manual Mode Only Available When Program  Is Not Running'
  937 = 'Metal Halide'
  493 = 'Metal Halide Lvl 1'
  494 = 'Metal Halide Lvl 2'
  495 = 'Metal Halide Lvl 3'
  585 = 'Minute'
  448 = 'Monday'
  602 = 'None'
  601 = 'Operator'
  946 = 'PID Equation Ref.'
  188 = 'Programs'
  938 = 'Ramp'
  387 = 'Rel. Humidity'
  200 = 'Saturday'
  491 = 'Schedule Sequence'
  600 = 'Service'
  385 = 'Setpoint'
  190 = 'Settings'
  321 = 'Setup Watering'
  197 = 'Start/Stop'
  410 = 'Stating A (Hour and Minute:'
  323 = 'Stating At :'
  304 = 'Stating at this time :'
  117 = 'Stating At:'
  939 = 'Step'
  929 = 'Sunday'
  944 = 'Td'
  399 = 'Temp Calibration Alarm'
  651 = 'Temp sensor 1'
  474 = 'Temp sensor 2'
  235 = 'Temp. Sensor '
  384 = 'Temperature'
  614 = 'Thursday'
  942 = 'Tn'
  375 = 'Tueday'
  322 = 'Tuesday'
  943 = 'Tv'
  198 = 'Users'
  659 = 'Valve Control \n(Integer 0-32767)'
  492 = 'Valve State'
  633 = 'Water on:'
  921 = 'Watering solenoid must be connected to Digital Out 9'
  858 = 'Watering solenoid must be connection to Digital Out 9'
  125 = 'Wednesday'
END_TEXTLIST

// ---- VISUs/HMI_MAIN.TcVIS
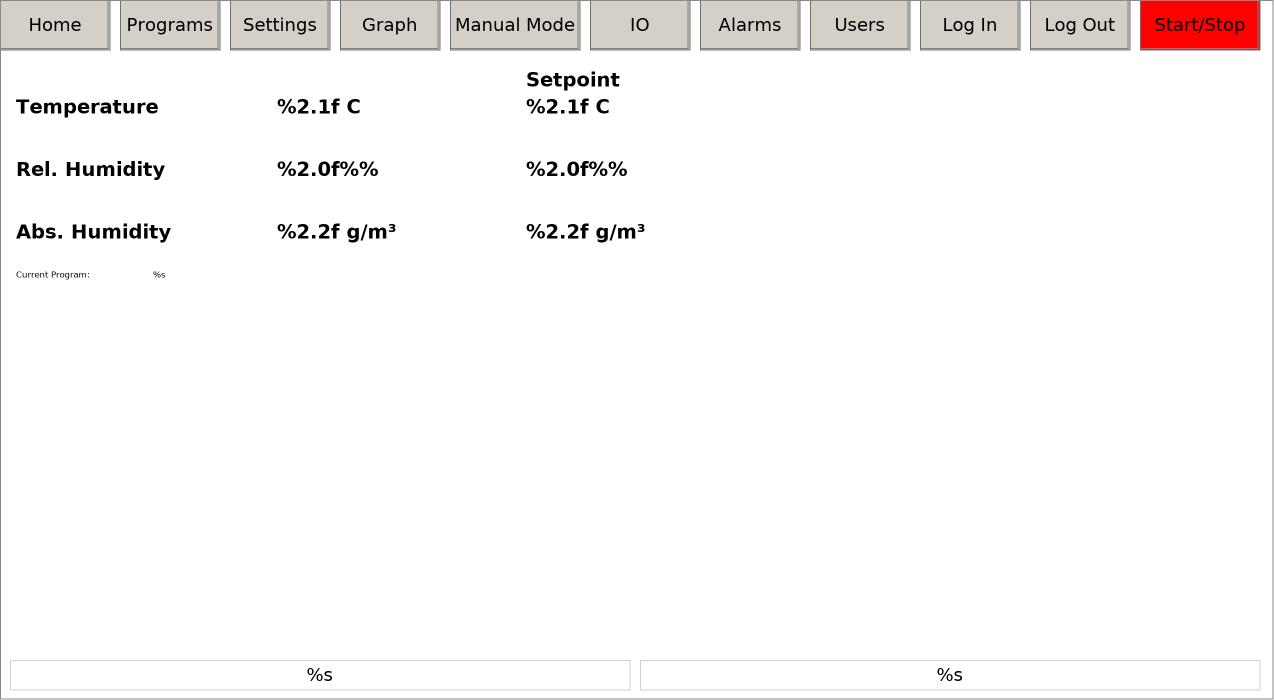
VISUALIZATION HMI_MAIN  // 1274x700
    Button (120,0 100x50), "Programs"
        OnMouseClick: FrameSelectionChange Selection=SelectedFrame=12e04cd0-f39d-4869-84a5-022adc51170e, Selection=1, GlobSel=AssignType=Directly, SelType=Locally
    Frame (0,60 1274x600)
        shows OverviewScreen()
        shows ProgramScreen()
        shows Settings()
        shows GraphScreen()
        shows ManualMode()
        shows IO()
        shows Alarms()
        shows Watering()
    Button (0,0 110x50), "Home"
        OnMouseClick: FrameSelectionChange Selection=SelectedFrame=12e04cd0-f39d-4869-84a5-022adc51170e, GlobSel=AssignType=Directly, SelType=Locally
    Button (230,0 100x50), "Settings"
        OnMouseClick: FrameSelectionChange Selection=SelectedFrame=12e04cd0-f39d-4869-84a5-022adc51170e, Selection=2, GlobSel=AssignType=Directly, SelType=Locally
    Button (340,0 100x50), "Graph"
        OnMouseClick: FrameSelectionChange Selection=SelectedFrame=12e04cd0-f39d-4869-84a5-022adc51170e, Selection=3, GlobSel=AssignType=Directly, SelType=Locally
    Button (450,0 130x50), "Manual Mode"
        OnMouseClick: FrameSelectionChange Selection=SelectedFrame=12e04cd0-f39d-4869-84a5-022adc51170e, Selection=4, GlobSel=AssignType=Directly, SelType=Locally
    Button (590,0 100x50), "IO"
        OnMouseClick: FrameSelectionChange Selection=SelectedFrame=12e04cd0-f39d-4869-84a5-022adc51170e, Selection=5, GlobSel=AssignType=Directly, SelType=Locally
    Button (700,0 100x50), "Alarms", colour toggle: GVL.bActiveAlarm
        OnMouseClick: FrameSelectionChange Selection=SelectedFrame=12e04cd0-f39d-4869-84a5-022adc51170e, Selection=6, GlobSel=AssignType=Directly, SelType=Locally
    Textfield (10,660 620x30), "%s", text variable: GVL.sAlarmText
    Textfield (640,660 620x30), "%s", text variable: GVL.sInfoText
    Button (920,0 100x50), "Log In"
        OnMouseClick: VisuUserMgmt Type=Login
    Button (1140,0 120x50), "Start/Stop", colour toggle: GVL.HMIPowerButton, input disabled if: GVL.manualMode
        OnMouseClick: toggle GVL.HMIPowerButton
    Button (810,0 100x50), "Users"
        OnMouseClick: VisuUserMgmt Type=OpenUserConfiguration
    Button (1030,0 100x50), "Log Out"
        OnMouseClick: VisuUserMgmt Type=Logout
END_VISUALIZATION

// ---- VISUs/OverviewScreen.TcVIS
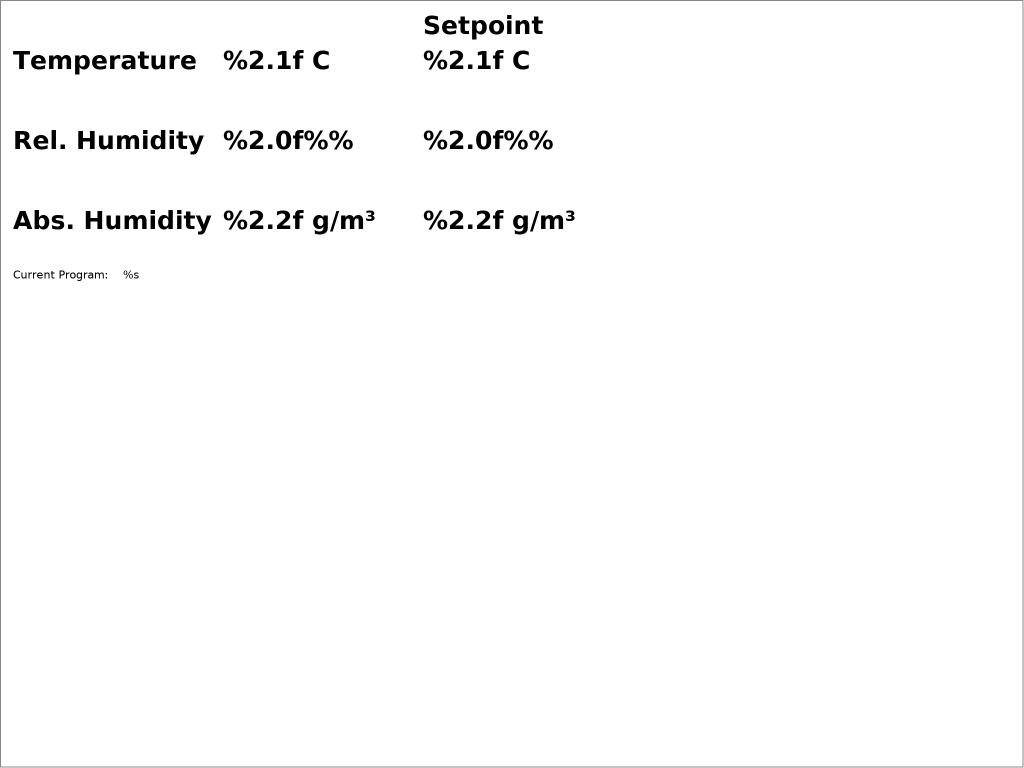
VISUALIZATION OverviewScreen  // 1024x768
    Rectangle (0,0 630x292)
    Textfield (220,40 200x40), "%2.1f C", text variable: GVL.Temp
    Textfield (420,40 200x40), "%2.1f C", text variable: GVL.TempSetpoint
    Label (10,40 200x40), "Temperature"
    Label (420,10 200x30), "Setpoint"
    Textfield (220,120 200x40), "%2.0f%%", text variable: GVL.Humidity
    Label (10,120 200x40), "Rel. Humidity"
    Textfield (120,260 120x30), "%s", text variable: GVL.CurrentProgramName
    Label (10,260 100x30), "Current Program:"
    Textfield (420,120 200x40), "%2.0f%%", text variable: GVL.HumiditySetpoint
    Textfield (220,200 200x40), "%2.2f g/m³", text variable: HumidityPID.AH
    Label (10,200 200x40), "Abs. Humidity"
    Textfield (420,200 200x40), "%2.2f g/m³", text variable: HumidityPID.AHSetpoint
END_VISUALIZATION

// ---- VISUs/GraphScreen.TcVIS
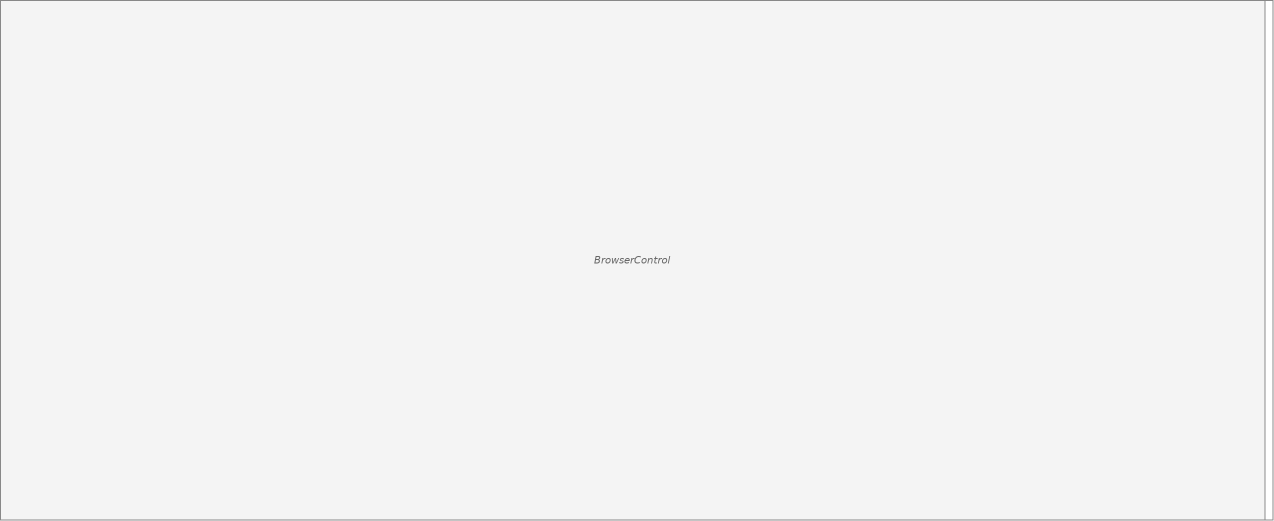
VISUALIZATION GraphScreen  // 1274x521
    BrowserControl (0,0 1265x520)
        p3734058945: GVL.graphURL
END_VISUALIZATION

// ---- VISUs/Settings.TcVIS
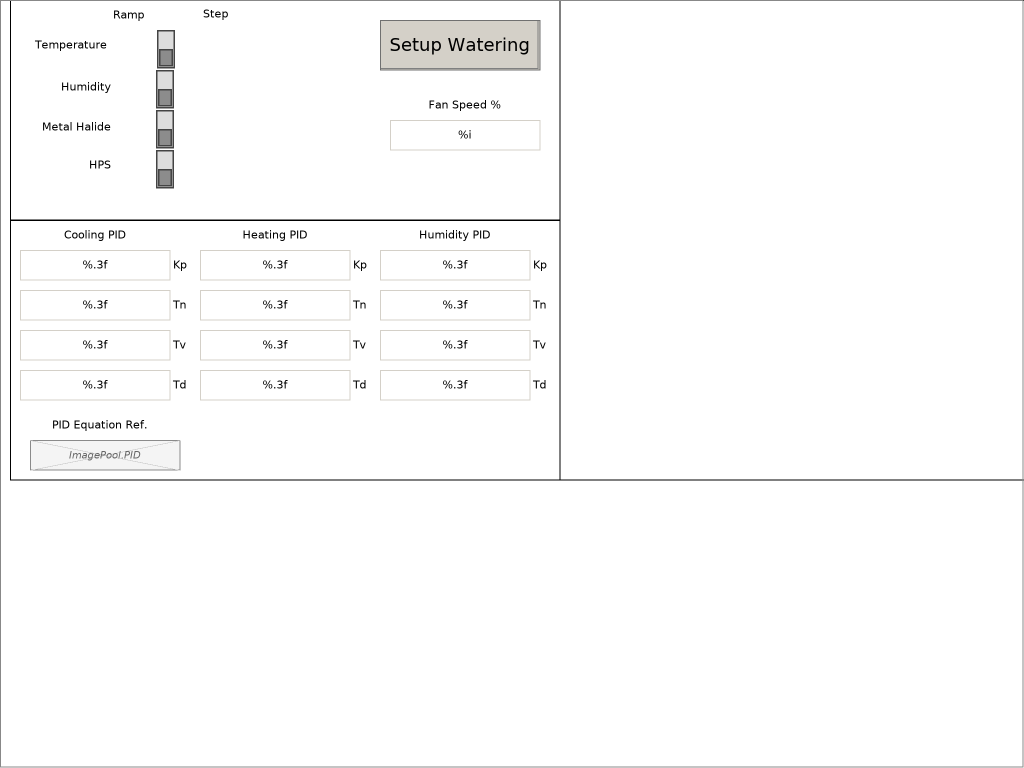
VISUALIZATION Settings  // 1024x768
    Rectangle (10,0 1025x480)
    Rectangle (10,0 550x220)
    Rectangle (10,220 550x260)
    DipSwitch (131,30 70x38), variable: GVL.TempStepmode, behaviour: TOGGLE, style: Switch-DipSwitch-Gray
    DipSwitch (130,110 70x38), variable: GVL.Light1Stepmode, behaviour: TOGGLE, style: Switch-DipSwitch-Gray
    Label (30,30 80x30), "Temperature"
    Label (0,112 114x30), "Metal Halide"
    Label (110,0 67x30), "Ramp"
    Label (200,0 49x28), "Step"
    Textfield (20,250 150x30), "%.3f", text variable: GVL.KpCooling
        OnMouseClick: write the text variable via VisuDialogs.Numpad, min 0
    Textfield (20,290 150x30), "%.3f", text variable: GVL.KiCooling
        OnMouseClick: write the text variable via VisuDialogs.Numpad, min 0
    Textfield (20,330 150x30), "%.3f", text variable: GVL.KvCooling
        OnMouseClick: write the text variable via VisuDialogs.Numpad, min 0
    Label (170,250 30x30), "Kp"
    Label (170,290 30x30), "Tn"
    Label (170,330 30x30), "Tv"
    Image (30,440 150x30), image: ImagePool.PID
    Textfield (20,370 150x30), "%.3f", text variable: GVL.KdCooling
        OnMouseClick: write the text variable via VisuDialogs.Numpad, min 0
    Label (170,370 30x30), "Td"
    Label (20,220 150x30), "Cooling PID"
    Label (0,410 200x30), "PID Equation Ref."
    Textfield (390,120 150x30), "%i", text variable: GVL.HMIFanSpeed
        OnMouseClick: write the text variable via VisuDialogs.Numpad, min 40, max 100
    Label (390,90 150x30), "Fan Speed %"
    Textfield (200,250 150x30), "%.3f", text variable: GVL.KpHeating
        OnMouseClick: write the text variable via VisuDialogs.Numpad, min 0
    Textfield (200,290 150x30), "%.3f", text variable: GVL.KiHeating
        OnMouseClick: write the text variable via VisuDialogs.Numpad, min 0
    Textfield (200,330 150x30), "%.3f", text variable: GVL.KvHeating
        OnMouseClick: write the text variable via VisuDialogs.Numpad, min 0
    Label (350,250 30x30), "Kp"
    Label (350,290 30x30), "Tn"
    Label (350,330 30x30), "Tv"
    Textfield (200,370 150x30), "%.3f", text variable: GVL.KdHeating
        OnMouseClick: write the text variable via VisuDialogs.Numpad, min 0
    Label (350,370 30x30), "Td"
    Label (200,220 150x30), "Heating PID"
    Textfield (380,250 150x30), "%.3f", text variable: GVL.KpHumidity
        OnMouseClick: write the text variable via VisuDialogs.Numpad, min 0
    Textfield (380,290 150x30), "%.3f", text variable: GVL.KiHumidity
        OnMouseClick: write the text variable via VisuDialogs.Numpad, min 0
    Textfield (380,330 150x30), "%.3f", text variable: GVL.KvHumidity
        OnMouseClick: write the text variable via VisuDialogs.Numpad, min 0
    Label (530,250 30x30), "Kp"
    Label (530,290 30x30), "Tn"
    Label (530,330 30x30), "Tv"
    Textfield (380,370 150x30), "%.3f", text variable: GVL.KdHumidity
        OnMouseClick: write the text variable via VisuDialogs.Numpad, min 0
    Label (530,370 30x30), "Td"
    Label (380,220 150x30), "Humidity PID"
    Label (0,72 114x30), "Humidity"
    DipSwitch (130,70 70x38), variable: GVL.HumidityStepmode, behaviour: TOGGLE, style: Switch-DipSwitch-Gray
    DipSwitch (130,150 70x38), variable: GVL.Light2Stepmode, behaviour: TOGGLE, style: Switch-DipSwitch-Gray
    Label (0,150 114x30), "HPS"
    Button (380,20 160x50), "Setup Watering"
        OnMouseClick: FrameSelectionChange Selection=Selection=-1, GlobSel=IndExpr=7, AssignDir=HMI_MAIN.GenElemInst_50, AssignType=Directly, SelType=Globally
END_VISUALIZATION

// ---- VISUs/ProgramScreen.TcVIS
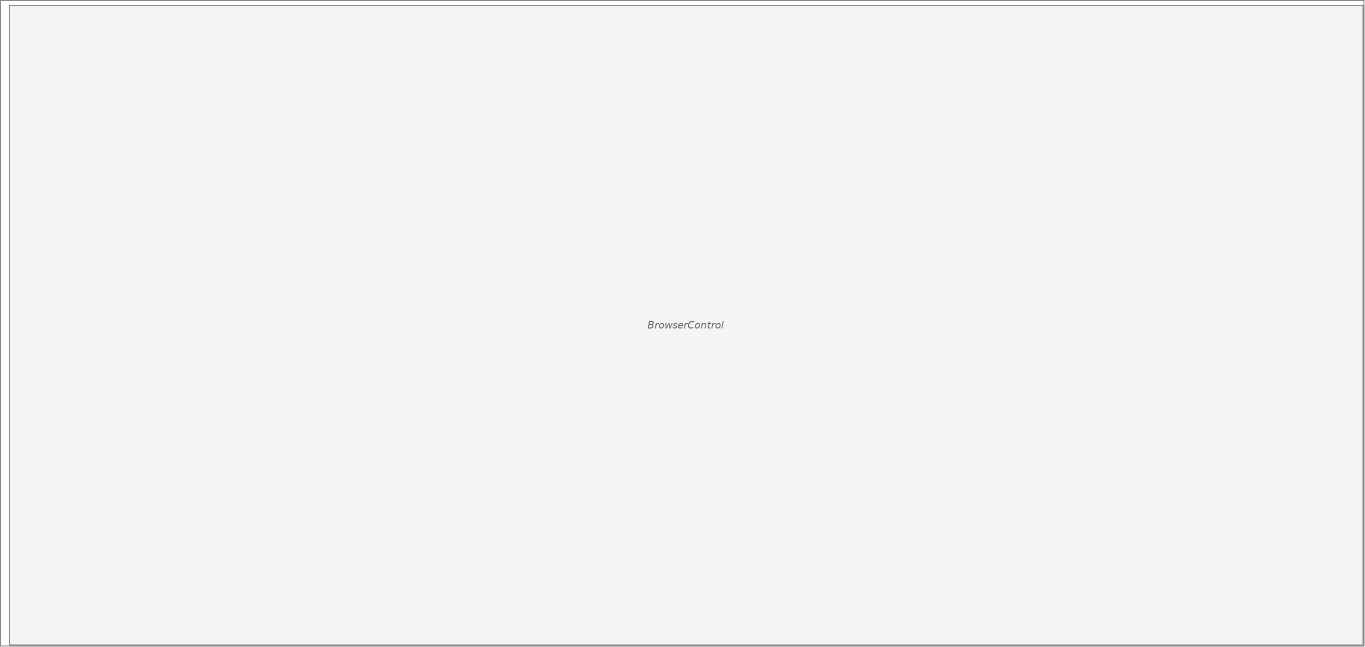
VISUALIZATION ProgramScreen  // 1365x647
    BrowserControl (9,5 1354x640)
        p3734058945: GVL.programURL
END_VISUALIZATION

// ---- VISUs/ManualMode.TcVIS
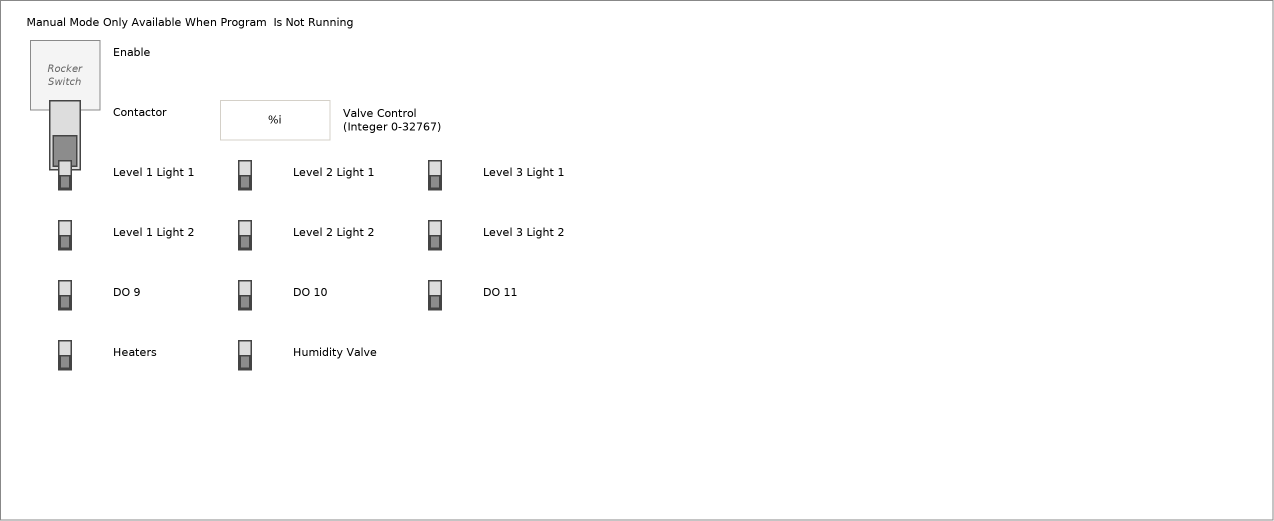
VISUALIZATION ManualMode  // 1274x521
    Label (10,10 360x25), "Manual Mode Only Available When Program Is Not Running"
    RockerSwitch (30,40 70x70), variable: GVL.manualMode, input disabled if: GVL.HMIPowerButton, behaviour: TOGGLE, style: Switch-RockerSwitch-Gray
    DipSwitch (30,100 70x70), variable: IO_VARS.ENABLE, behaviour: TOGGLE, style: Switch-DipSwitch-Gray
    Label (110,40 80x25), "Enable"
    Label (110,100 80x25), "Contactor"
    Label (110,160 110x25), "Level 1 Light 1"
    Label (110,220 110x25), "Level 1 Light 2"
    Textfield (220,100 110x40), "%i", text variable: IO_VARS.GLYCOL_VALVE
        OnMouseClick: write the text variable via VisuDialogs.Numpad, min 0, max 32767
    Label (340,100 100x40), "Valve Control (Integer 0-32767)"
    DipSwitch (30,160 70x30), variable: IO_VARS.MH1, behaviour: TOGGLE, style: Switch-DipSwitch-Gray
    DipSwitch (30,220 70x30), variable: IO_VARS.HPS1, behaviour: TOGGLE, style: Switch-DipSwitch-Gray
    Label (290,160 110x25), "Level 2 Light 1"
    Label (290,220 110x25), "Level 2 Light 2"
    DipSwitch (210,160 70x30), variable: IO_VARS.MH2, behaviour: TOGGLE, style: Switch-DipSwitch-Gray
    DipSwitch (210,220 70x30), variable: IO_VARS.HPS2, behaviour: TOGGLE, style: Switch-DipSwitch-Gray
    Label (480,160 110x25), "Level 3 Light 1"
    Label (480,220 110x25), "Level 3 Light 2"
    DipSwitch (400,160 70x30), variable: IO_VARS.MH3, behaviour: TOGGLE, style: Switch-DipSwitch-Gray
    DipSwitch (400,220 70x30), variable: IO_VARS.HPS3, behaviour: TOGGLE, style: Switch-DipSwitch-Gray
    Label (110,280 110x25), "DO 9"
    DipSwitch (30,280 70x30), variable: IO_VARS.AUX1, behaviour: TOGGLE, style: Switch-DipSwitch-Gray
    Label (290,280 110x25), "DO 10"
    DipSwitch (210,280 70x30), variable: IO_VARS.AUX2, behaviour: TOGGLE, style: Switch-DipSwitch-Gray
    Label (480,280 110x25), "DO 11"
    DipSwitch (400,280 70x30), variable: IO_VARS.AUX3, behaviour: TOGGLE, style: Switch-DipSwitch-Gray
    Label (110,340 110x25), "Heaters"
    DipSwitch (30,340 70x30), variable: IO_VARS.HEATERS, behaviour: TOGGLE, style: Switch-DipSwitch-Gray
    Label (290,340 110x25), "Humidity Valve"
    DipSwitch (210,340 70x30), variable: IO_VARS.HUMVALVE, behaviour: TOGGLE, style: Switch-DipSwitch-Gray
END_VISUALIZATION

// ---- VISUs/IO.TcVIS
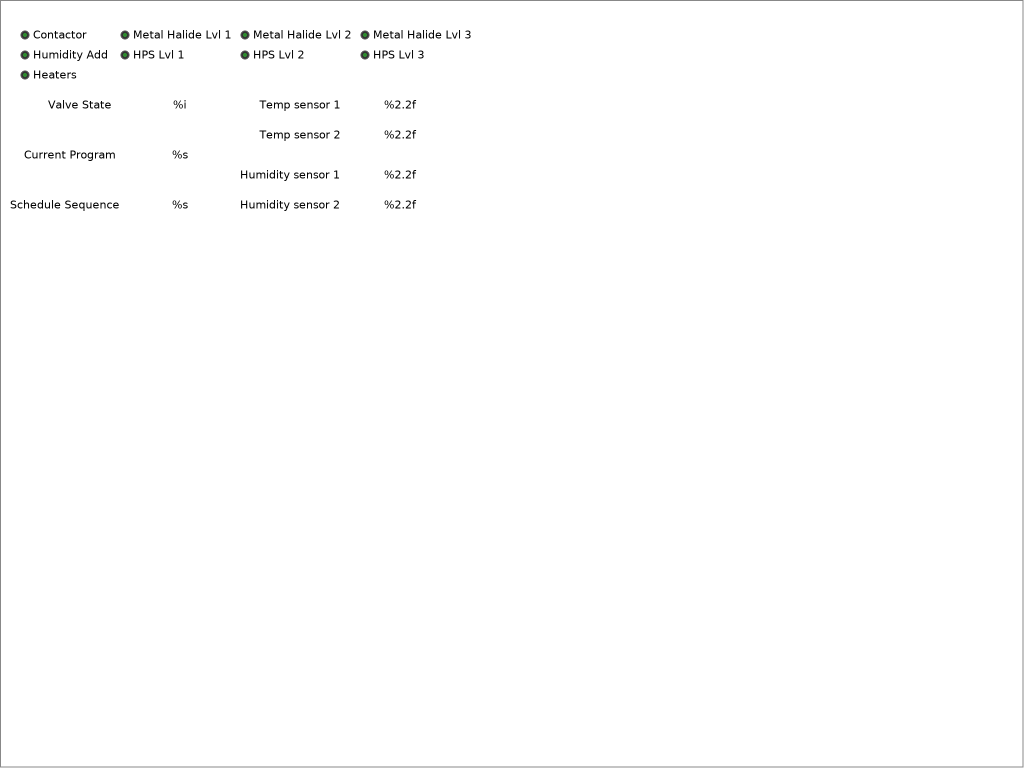
VISUALIZATION IO  // 1024x768
    Lamp1 (20,30 10x10), variable: IO_VARS.ENABLE, style: Lamp-Lamp1-Green
    Label (30,20 100x30), "Contactor"
    Textfield (130,140 100x30), "%s", text variable: GVL.CurrentProgramName
    Label (20,140 100x30), "Current Program"
    Label (10,190 110x30), "Schedule Sequence"
    Textfield (130,190 100x30), "%s", text variable: GVL.ScheduleSequence
    Textfield (130,90 100x30), "%i", text variable: GVL.iTempControl
    Label (30,90 100x30), "Valve State"
    Lamp1 (120,30 10x10), variable: IO_VARS.MH1, style: Lamp-Lamp1-Green
    Label (130,20 100x30), "Metal Halide Lvl 1"
    Lamp1 (240,30 10x10), variable: IO_VARS.MH2, style: Lamp-Lamp1-Green
    Label (250,20 100x30), "Metal Halide Lvl 2"
    Lamp1 (360,30 10x10), variable: IO_VARS.MH3, style: Lamp-Lamp1-Green
    Label (370,20 100x30), "Metal Halide Lvl 3"
    Lamp1 (120,50 10x10), variable: IO_VARS.HPS1, style: Lamp-Lamp1-Green
    Label (130,40 100x30), "HPS Lvl 1"
    Lamp1 (240,50 10x10), variable: IO_VARS.HPS2, style: Lamp-Lamp1-Green
    Label (250,40 100x30), "HPS Lvl 2"
    Lamp1 (360,50 10x10), variable: IO_VARS.HPS3, style: Lamp-Lamp1-Green
    Label (370,40 100x30), "HPS Lvl 3"
    Label (30,40 100x30), "Humidity Add"
    Lamp1 (20,50 10x10), variable: IO_VARS.HUMVALVE, style: Lamp-Lamp1-Green
    Label (30,60 100x30), "Heaters"
    Lamp1 (20,70 10x10), variable: IO_VARS.HEATERS, style: Lamp-Lamp1-Green
    Label (250,90 100x30), "Temp sensor 1"
    Textfield (350,90 100x30), "%2.2f", text variable: GVL.Temp
    Label (250,120 100x30), "Temp sensor 2"
    Textfield (350,120 100x30), "%2.2f", text variable: GVL.Temp2
    Label (230,160 120x30), "Humidity sensor 1"
    Textfield (350,160 100x30), "%2.2f", text variable: GVL.Humidity
    Label (230,190 120x30), "Humidity sensor 2"
    Textfield (350,190 100x30), "%2.2f", text variable: GVL.Humidity2
END_VISUALIZATION

// ---- VISUs/Alarms.TcVIS
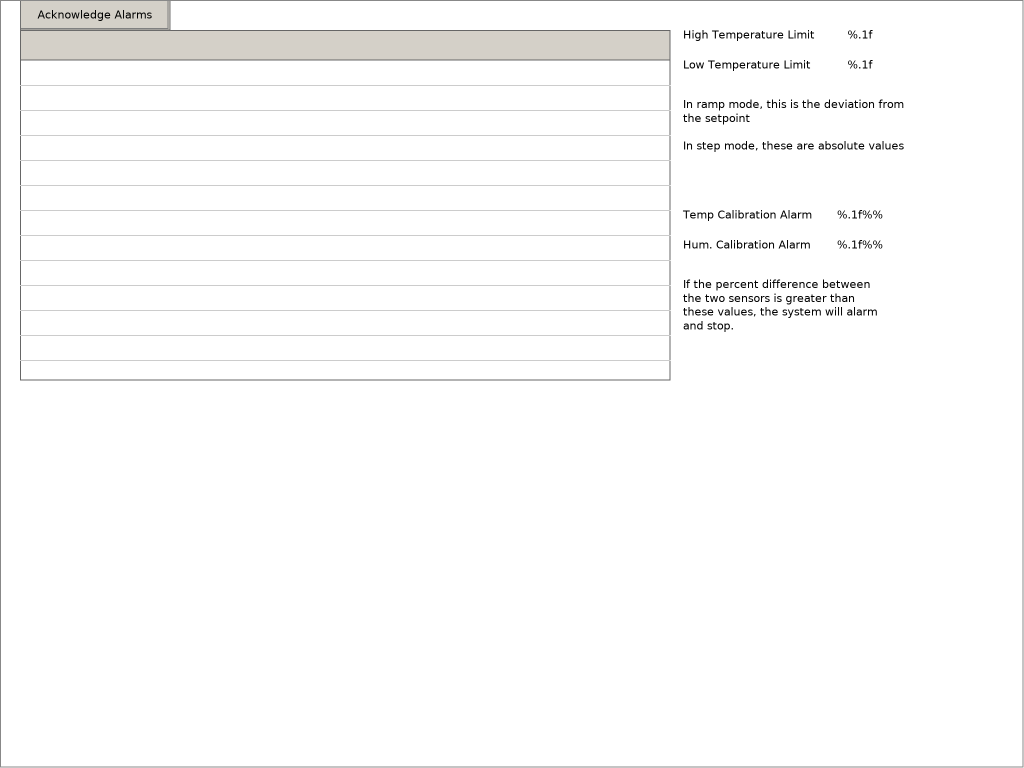
VISUALIZATION Alarms  // 1024x768
    Table (20,30 650x350), data array: GVL.aAlarms
        p511219082: Alarm Note
        p1892666644: GVL.aAlarms[INDEX].sAlarmText
        p2232123230: Date & Time
        p3854506369: GVL.aAlarms[INDEX].dtTime
    Textfield (810,20 100x30), "%.1f", text variable: GVL.TempAlarmHigh
        OnMouseClick: write the text variable via VisuDialogs.Numpad, min -10, max 50
    Label (680,20 150x30), "High Temperature Limit"
    Textfield (810,50 100x30), "%.1f", text variable: GVL.TempAlarmLow
        OnMouseClick: write the text variable via VisuDialogs.Numpad, min -10, max 50
    Label (680,50 150x30), "Low Temperature Limit"
    Button (20,0 150x30), "Acknowledge Alarms", colour toggle: GVL.bActiveAlarm
        OnMouseClick: execute { GVL.bActiveAlarm:=FALSE; }
    Textfield (680,90 260x70), "In ramp mode, this is the deviation from the setpoint In step mode, these are absolute values"
    Textfield (810,200 100x30), "%.1f%%", text variable: GVL.TempCalibrationLimit
        OnMouseClick: write the text variable via Default, min 1, max 100
    Label (680,200 150x30), "Temp Calibration Alarm"
    Textfield (810,230 100x30), "%.1f%%", text variable: GVL.HumCalibrationLimit
        OnMouseClick: write the text variable via VisuDialogs.Numpad, min 1, max 100
    Label (680,230 150x30), "Hum. Calibration Alarm"
    Textfield (680,270 260x70), "If the percent difference between the two sensors is greater than these values, the system will alarm and stop."
END_VISUALIZATION

// ---- VISUs/Watering.TcVIS
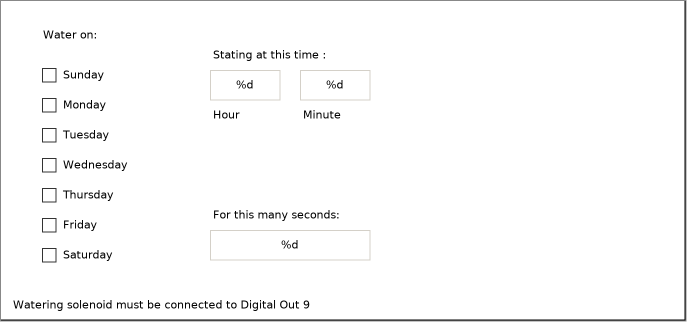
VISUALIZATION Watering  // 687x322
    Rectangle (0,0 685x320)
    Checkbox (40,60 150x30), "Sunday", variable: GVL.wateringDays[0]
    Checkbox (40,90 150x30), "Monday", variable: GVL.wateringDays[1]
    Checkbox (40,120 150x30), "Tuesday", variable: GVL.wateringDays[2]
    Checkbox (40,150 150x30), "Wednesday", variable: GVL.wateringDays[3]
    Checkbox (40,180 150x30), "Thursday", variable: GVL.wateringDays[4]
    Checkbox (40,210 150x30), "Friday", variable: GVL.wateringDays[5]
    Checkbox (40,240 150x30), "Saturday", variable: GVL.wateringDays[6]
    Textfield (210,70 70x30), "%d", text variable: GVL.HMIWateringStartHour
        OnMouseClick: write the text variable via VisuDialogs.Numpad, min 0, max 23, title 'Hour 0-23'
    Textfield (300,70 70x30), "%d", text variable: GVL.HMIWateringStartMinute
        OnMouseClick: write the text variable via VisuDialogs.Numpad, min 0, max 59, title 'Minute 0-59'
    Textfield (210,230 160x30), "%d", text variable: GVL.HMIWateringTimeSeconds
        OnMouseClick: write the text variable via VisuDialogs.Numpad, min 0, max 86400, title 'Duration (seconds)'
    Label (40,20 60x30), "Water on:"
    Label (210,40 180x30), "Stating at this time :"
    Label (210,200 140x30), "For this many seconds:"
    Label (210,100 40x30), "Hour"
    Label (300,100 80x30), "Minute"
    Label (10,290 320x30), "Watering solenoid must be connected to Digital Out 9"
END_VISUALIZATION
